Staubli VAL3: MFX_ROB_17.pjx

--- MFX_ROB_17.pjx ---
Parameters version=s7.9.1 stackSize=5000 millimeterUnit=true
Program file=checkAtPark.pgx
Program file=display.pgx
Program file=displayMessage.pgx
Program file=displayMessage1.pgx
Program file=displayMessage2.pgx
Program file=displayMessage3.pgx
Program file=displayMessage4.pgx
Program file=displayMessage5.pgx
Program file=displayMessage6.pgx
Program file=displayMessage7.pgx
Program file=displayMessage8.pgx
Program file=displayMessage9.pgx
Program file=initialize.pgx
Program file=initializeRobot.pgx
Program file=iocWriteBack.pgx
Program file=main.pgx
Program file=makePntAZELRA.pgx
Program file=mnuAdjTargetPnt.pgx
Program file=mnuEnterIPVals.pgx
Program file=mnuEnterTCPVals.pgx
Program file=mnuGetTCP.pgx
Program file=mnuGlobalSpeed.pgx
Program file=mnuMotionMenu.pgx
Program file=mnuMoveTargPnt.pgx
Program file=mnuMoveToPark.pgx
Program file=mnuSetTargetPts.pgx
Program file=mnuTeachCube.pgx
Program file=mnuTeachCyl.pgx
Program file=mnuTeachFrame.pgx
Program file=mnuTeachIP.pgx
Program file=mnuTeachMenu.pgx
Program file=mnuTeachPark.pgx
Program file=mnuTeachParkTop.pgx
Program file=mnuTeachSphere.pgx
Program file=mnuTeachStayClr.pgx
Program file=mnuTeachTCP.pgx
Program file=mnuTeachTCP4pnt.pgx
Program file=mnuTeachTCPptr.pgx
Program file=mnuTestSimESTOP.pgx
Program file=mnuUtility.pgx
Program file=movTargetPoint.pgx
Program file=movToPark.pgx
Program file=movToParkTop.pgx
Program file=readme.pgx
Program file=remCalcHere.pgx
Program file=remCalcHereSph.pgx
Program file=remCmdHandler.pgx
Program file=remDisableArm.pgx
Program file=remEnableArm.pgx
Program file=remEnableRem.pgx
Program file=remErrArgs.pgx
Program file=remErrBufferAdd.pgx
Program file=remErrBufferGet.pgx
Program file=remErrBusy.pgx
Program file=remErrCmd.pgx
Program file=remErrConfig.pgx
Program file=remErrFar.pgx
Program file=remErrInvalid.pgx
Program file=remErrManual.pgx
Program file=remErrNum.pgx
Program file=remErrPower.pgx
Program file=remErrPPTimeout.pgx
Program file=remErrRemoteKey.pgx
Program file=remErrTimeout.pgx
Program file=remErrZone.pgx
Program file=remGetArmStat.pgx
Program file=remGetDMOV.pgx
Program file=remGetESTOP.pgx
Program file=remGetHeartbeat.pgx
Program file=remGetHere.pgx
Program file=remGetHereSph.pgx
Program file=remGetIP.pgx
Program file=remGetIPVals.pgx
Program file=remGetJoints.pgx
Program file=remGetMaxA.pgx
Program file=remGetMaxDist.pgx
Program file=remGetMaxRV.pgx
Program file=remGetMaxV.pgx
Program file=remGetMode.pgx
Program file=remGetOneHere.pgx
Program file=remGetPPS.pgx
Program file=remGetRem.pgx
Program file=remGetRobotMode.pgx
Program file=remGetStagePos.pgx
Program file=remGetTCPVals.pgx
Program file=remGetWorld.pgx
Program file=remGetnGlobal.pgx
Program file=remMovAZELRA.pgx
Program file=remMovAxis.pgx
Program file=remMovBase.pgx
Program file=remMovHandler.pgx
Program file=remMovJoint.pgx
Program file=remMovJointAxis.pgx
Program file=remMovPoint.pgx
Program file=remMovSph.pgx
Program file=remMovSphAxis.pgx
Program file=remMovXYZ.pgx
Program file=remSetHeartbeat.pgx
Program file=remSetIP.pgx
Program file=remSetIPVals.pgx
Program file=remSetMaxA.pgx
Program file=remSetMaxDist.pgx
Program file=remSetMaxRV.pgx
Program file=remSetMaxV.pgx
Program file=remSetMode.pgx
Program file=remSetPPS.pgx
Program file=remSetStagePos.pgx
Program file=remSetTCPVals.pgx
Program file=remSetnGlobal.pgx
Program file=remTest.pgx
Program file=remTransIP.pgx
Program file=start.pgx
Program file=stop.pgx
Program file=tskCollision.pgx
Program file=tskHaltMoveMon.pgx
Program file=tskInterlocks.pgx
Program file=tskMonitorZone.pgx
Program file=tskRemControl1.pgx
Program file=tskSimESTOP.pgx
Data file=MFX_ROB_17.dtx
Library alias=io path=Disk://io/io.pjx autoload=true password=
Library alias=TCP4 path=Disk://calcTool4pEn/calcTool4pEn.pjx autoload=true password=
Library alias=MON path=Disk://monitorAreaEn/monitorAreaEn.pjx autoload=true password=

--- MFX_ROB_17.dtx ---
public bool bCubeStep1
public bool bCylinderStep1
bool bESTOPactive
public bool bEnableMonitor
public bool bInsideCube
public bool bInsideCylinder
public bool bInsideSphere
bool bKillRemControl
bool bMoveLinear = true
public bool bRemControlON
bool bRemMotionBusy
public bool bSetCubeXYZ
public bool bSetCylinderRZ
public bool bSetSphereRad
bool bSimESTOPOn
bool bSimulateESTOP
public bool bSphereStep1
public bool bStopAllMonitor = true
public bool bStopMotion
public bool bWatchForHalt
public bool bWorldFrameView = true
dio dCollisionSens = {link=usrIn0}
frame fIP1 = {fatherId=fIPoriginal[0]}
public frame fIP2 = {fatherId=fIPoriginal[0]}
frame fIPoriginal = {x=-1.16, y=-7.997692, z=1599.75028, rx=-90.079848, ry=0.325339, rz=-0.147005, fatherId=world[0]}
public jointRx jPark = {j1=89.588014, j2=-47.40785, j3=113.936199, j4=-0.155325, j5=-66.458795, j6=0.148711}
jointRx jParkTop = {j1=88.830052, j2=-90.553253, j3=149.996753, j4=-0.166481, j5=-59.375003, j6=0.928419}
mdesc mDefault = {accel=20, vel=20, decel=20, blend=off}
public mdesc mGlobalSpeed = {accel=20, vel=20, decel=20, blend=off}
mdesc mMdesc
public mdesc mSafeSlow = {accel=15, vel=20, decel=15, blend=off}
num nAccFast = 60
num nAccMedium = 40
num nAccSlow = 20
num nAdjPntMoveTol = 25
num nAzHere = -0.0000183783
num nColision = 1
num nDistXCube
num nDistYCube
num nDistZCube
num nDistZCylinder
num nElHere = 44.997695
num nErrBufferSize = 10
num nErrNext
num nErrNow
num nHeartbeat = 4344
num nIP1Azimuth[20]
  [1] = 45
  [2] = -45
  [3] = 45
  [4] = -45
  [5] = 9.38
  [6] = 7.44
  [7] = 17.53
  [8] = 48.36
  [9] = 142.53
  [10] = 140.2
  [11] = 145.08
  [12] = 142.4
  [13] = 142.23
  [14] = 144.96
  [15] = 106.35
  [16] = 100.36
  [17] = 19.8
  [18] = 8.88
  [19] = 23.034688
num nIP1Elevation[20]
  [3] = -45
  [4] = -45
  [5] = 21.19
  [6] = 39.23
  [9] = 37.74
  [10] = 30.33
  [11] = 44.59
  [12] = 42.45
  [13] = 38.39
  [14] = 44.81
  [15] = 29.56
  [16] = 45.35
  [17] = 29.88
  [18] = 12.25
  [19] = 8.727177
num nIP1Number = 1
num nIP1Radius[20]
  [1] = 600
  [2] = 600
  [3] = 600
  [4] = 600
  [5] = 1000
  [6] = 1000
  [7] = 300
  [8] = 250
  [9] = 300
  [10] = 300
  [11] = 300
  [12] = 300
  [13] = 300
  [14] = 300
  [15] = 300
  [16] = 300
  [17] = 100
  [18] = 200
  [19] = 857.27654
num nIP2Azimuth[20]
  [0] = 15
  [2] = -128.927
num nIP2Elevation[20]
  [0] = 20
  [2] = 79.165
num nIP2Number = 2
num nIP2Radius[20]
  [0] = 300
  [1] = 600
  [2] = 123.321
  [5] = 1000
num nIPNumber = -1
num nIdxAdjTargetPt = 291
num nIdxArmCalCheck = 31
num nIdxArmPowerOn = 181
num nIdxESTOPCheck = 121
num nIdxEnterIP = 341
num nIdxEnterTCP = 321
public num nIdxFrm1of5 = 131
public num nIdxFrm2of5 = 141
public num nIdxFrm3of5 = 151
public num nIdxFrm4of5 = 161
public num nIdxFrm5of5 = 171
num nIdxGetTCP = 351
public num nIdxMainMenu = 1
public num nIdxMotionMenu = 271
num nIdxMoveTargPt = 281
num nIdxMoveToPark = 311
num nIdxParkCheck = 41
public num nIdxPtrVerify
num nIdxRemControl = 321
public num nIdxResolution
public num nIdxSetCubeXYZ = 211
public num nIdxSetCylRZ = 231
num nIdxSetSpeeds = 181
public num nIdxSetSphRad = 251
num nIdxSetTargetPt = 261
public num nIdxStyClr = 61
public num nIdxTCP1of4 = 81
public num nIdxTCP2of4 = 91
public num nIdxTCP3of4 = 101
public num nIdxTCP4Point
public num nIdxTCP4of4 = 111
public num nIdxTeachClear
public num nIdxTeachCube = 201
public num nIdxTeachCyl = 221
num nIdxTeachIP = 331
public num nIdxTeachMenu = 11
public num nIdxTeachPARK = 51
num nIdxTeachPARKT = 371
public num nIdxTeachSph = 241
public num nIdxTeachTCP = 21
num nIdxUtilMenu2 = 301
num nIdxUtilityMenu = 71
num nMaxAccel = 50
num nMaxDist = 1000
num nMaxLoginTries = 3
num nMaxRVelo = 20
num nMaxVelo = 100
num nMovArgs
num nNumberCube
num nNumberCylinder
num nNumberSphere
num nPPS
num nParkTolerance = 50
num nRHere = 565.684578
num nRXHere = 0.0101053
num nRYHere = 0.000281961
num nRZHere = 0.00483895
num nRadiusCylinder
num nRadiusSphere
num nRemoteTimeout = 30
num nResolution[4]
  [0] = 0.001
  [1] = 0.01
  [2] = 0.1
  [3] = 1
num nRobotMode = 1
num nSelection = 1
num nStagePos
num nStagePosOK
num nVelFast = 60
num nVelMedium = 40
num nVelSlow = 20
num nXHere = -0.00012746
num nYHere = 399.983479
num nZHere = 400.0163407
num nZoneWatchTol = 25
public pointRx pCellReference = {shoulder=righty, elbow=epositive, wrist=wpositive, fatherId=world[0]}
pointRx pIP1NullPoint = {shoulder=sfree, elbow=efree, wrist=wfree, fatherId=fIP1[0]}
pointRx pIP1Point[20]
  [0] = {x=73, y=424, z=417, rx=-45, ry=-172, rz=-7, shoulder=sfree, elbow=efree, wrist=wfree, fatherId=fIP1[0]}
  [1] = {x=145, y=424, z=398, rx=-46, ry=-166, rz=-14, shoulder=sfree, elbow=efree, wrist=wfree, fatherId=fIP1[0]}
  [2] = {x=272, y=424, z=325, rx=-52, ry=-152, rz=-30, shoulder=sfree, elbow=efree, wrist=wfree, fatherId=fIP1[0]}
  [3] = {x=325, y=424, z=272, rx=-57, ry=-147, rz=-40, shoulder=sfree, elbow=efree, wrist=wfree, fatherId=fIP1[0]}
  [4] = {x=294, y=424, z=305, rx=-54, ry=-150, rz=-34, shoulder=sfree, elbow=efree, wrist=wfree, fatherId=fIP1[0]}
  [5] = {fatherId=fIP1[0]}
  [6] = {fatherId=fIP1[0]}
  [7] = {x=145, y=424, z=398, rx=-46, ry=-166, rz=-14, fatherId=fIP1[0]}
  [8] = {fatherId=fIP1[0]}
  [9] = {x=272, y=424, z=325, rx=-52, ry=-152, rz=-30, fatherId=fIP1[0]}
  [10] = {fatherId=fIP1[0]}
  [11] = {fatherId=fIP1[0]}
  [12] = {x=325, y=424, z=272, rx=-57, ry=-147, rz=-40, fatherId=fIP1[0]}
  [13] = {x=294, y=424, z=305, rx=-54, ry=-150, rz=-34, fatherId=fIP1[0]}
  [14] = {fatherId=fIP1[0]}
  [15] = {fatherId=fIP1[0]}
  [16] = {fatherId=fIP1[0]}
  [17] = {fatherId=fIP1[0]}
  [18] = {fatherId=fIP1[0]}
  [19] = {y=500, rx=90, rz=-180, fatherId=fIP1[0]}
pointRx pIP2NullPoint = {fatherId=fIP2[0]}
pointRx pIP2Point[20]
  [0] = {shoulder=sfree, elbow=efree, wrist=wfree, fatherId=fIP2[0]}
  [1] = {x=300, y=424.264069, z=300, rx=125.26439, ry=-30, rz=-35.26439, shoulder=sfree, elbow=efree, wrist=wfree, fatherId=fIP2[0]}
  [2] = {x=-300, y=424.264069, z=300, rx=125.26439, ry=30, rz=35.26439, shoulder=sfree, elbow=efree, wrist=wfree, fatherId=fIP2[0]}
  [3] = {x=300, y=-424.264069, z=300, rx=-125.26439, ry=-30, rz=35.26439, shoulder=sfree, elbow=efree, wrist=wfree, fatherId=fIP2[0]}
  [4] = {x=-300, y=-424.264069, z=300, rx=-125.26439, ry=30, rz=-35.26439, shoulder=sfree, elbow=efree, wrist=wfree, fatherId=fIP2[0]}
  [5] = {shoulder=sfree, elbow=efree, wrist=wfree, fatherId=fIP2[0]}
  [6] = {shoulder=sfree, elbow=efree, wrist=wfree, fatherId=fIP2[0]}
  [7] = {shoulder=sfree, elbow=efree, wrist=wfree, fatherId=fIP2[0]}
  [8] = {shoulder=sfree, elbow=efree, wrist=wfree, fatherId=fIP2[0]}
  [9] = {shoulder=sfree, elbow=efree, wrist=wfree, fatherId=fIP2[0]}
  [10] = {shoulder=sfree, elbow=efree, wrist=wfree, fatherId=fIP2[0]}
  [11] = {shoulder=sfree, elbow=efree, wrist=wfree, fatherId=fIP2[0]}
  [12] = {shoulder=sfree, elbow=efree, wrist=wfree, fatherId=fIP2[0]}
  [13] = {shoulder=sfree, elbow=efree, wrist=wfree, fatherId=fIP2[0]}
  [14] = {shoulder=sfree, elbow=efree, wrist=wfree, fatherId=fIP2[0]}
  [15] = {shoulder=sfree, elbow=efree, wrist=wfree, fatherId=fIP2[0]}
  [16] = {shoulder=sfree, elbow=efree, wrist=wfree, fatherId=fIP2[0]}
  [17] = {shoulder=sfree, elbow=efree, wrist=wfree, fatherId=fIP2[0]}
  [18] = {shoulder=sfree, elbow=efree, wrist=wfree, fatherId=fIP2[0]}
  [19] = {shoulder=sfree, elbow=efree, wrist=wfree, fatherId=fIP2[0]}
pointRx pMoveIP1Target = {fatherId=fIP1[0]}
pointRx pMoveIP2Target = {shoulder=sfree, elbow=efree, wrist=wfree, fatherId=fIP2[0]}
pointRx pMoveTarget = {shoulder=sfree, elbow=efree, wrist=wfree, fatherId=world[0]}
pointRx pNullPosition = {fatherId=world[0]}
pointRx pOriginCube = {fatherId=world[0]}
pointRx pOriginCylinder = {fatherId=world[0]}
pointRx pOriginSphere = {fatherId=world[0]}
pointRx teste[4]
  [0] = {x=7, y=243, z=26, rx=-4.03658e-18, ry=-79, rz=-9.47474e-33, shoulder=sfree, elbow=efree, wrist=wfree, fatherId=fIP1[0]}
  [1] = {x=17, y=243, z=28, rx=4.437099e-14, ry=-79.999286, rz=0.00497464, fatherId=fIP1[0]}
  [2] = {y=400, z=400, rx=0.01, ry=-2.827901e-23, rz=0.00516647, fatherId=fIP1[0]}
  [3] = {fatherId=fIP1[0]}
sio sioIOCclient = {link=Socket\MFX}
string sErrBuffer[10]
string sIOCCommand
string sIOCPassword = "USERPASSWORD"
string sIOCUserName = "CS8LOGIN"
string sIOCValue
string sIP1TargName[20]
  [0] = "v"
  [1] = "a"
  [2] = "sto 1"
  [3] = "ybco104"
  [4] = "cool oi"
  [5] = "magpeak2"
  [6] = "IP1 Point6 Name"
  [7] = "IP1 Point7 Name"
  [8] = "IP1 Point8 Name"
  [9] = "IP1 Point9 Name"
  [10] = "IP1 Point10 Name"
  [11] = "IP1 Point11 Name"
  [12] = "IP1 Point12 Name"
  [13] = "IP1 Point13 Name"
  [14] = "IP1 Point14 Name"
  [15] = "IP1 Point15 Name"
  [16] = "IP1 Point16 Name"
  [17] = "IP1 Point17 Name"
  [18] = "IP1 Point18 Name"
  [19] = "IP1 Point19 Name"
string sIP2TargName[20]
  [0] = "TestTeachPoint0"
  [1] = "IP2 Point1 Name"
  [2] = "IP2 Point2 Name"
  [3] = "IP2 Point3 Name"
  [4] = "IP2 Point4 Name"
  [5] = "a"
  [6] = "IP2 Point6 Name"
  [7] = "IP2 Point7 Name"
  [8] = "IP2 Point8 Name"
  [9] = "IP2 Point9 Name"
  [10] = "IP2 Point10 Name"
  [11] = "IP2 Point11 Name"
  [12] = "IP2 Point12 Name"
  [13] = "IP2 Point13 Name"
  [14] = "IP2 Point14 Name"
  [15] = "IP2 Point15 Name"
  [16] = "IP2 Point16 Name"
  [17] = "IP2 Point17 Name"
  [18] = "IP2 Point18 Name"
  [19] = "IP2 Point19 Name"
string sMenuBottomLine[53]
  [0] = " Tch. Mot. Util ---- ---- ---- ---- Stop"
  [1] = " Pnts IPCS Park ParkT TCP Zone  --- Ret."
  [2] = "RefP 4Pnt DEnt ---- ---- ---- ---- Ret."
  [3] = "---- ---- ---- Stop ---- ---- ---- Ret."
  [4] = "Cont ---- ---- Mov. ---- ---- ---- Ret."
  [5] = "Save ---- ---- ---- ---- ---- ---- Ret."
  [6] = "Cube Cyl. Sph. ---- ---- ---- ---- Ret."
  [7] = "Init Park Enbl Spds RemC TCP. ---- Ret."
  [8] = "Next ---- ---- ---- ---- ---- ---- Abrt"
  [9] = "Next ---- ---- ---- ---- ---- ---- Abrt"
  [10] = "Next ---- ---- ---- ---- ---- ---- Abrt"
  [11] = "Tch. ---- ---- ---- ---- ---- ---- Abrt"
  [12] = "Cont ---- ---- ---- ---- ---- ---- Abrt"
  [13] = "Next ---- Togl ---- ---- ---- ---- Abrt"
  [14] = "Next ---- ---- ---- ---- ---- ---- Abrt"
  [15] = "Next ---- ---- ---- ---- ---- ---- Abrt"
  [16] = "Next ---- ---- ---- ---- ---- ---- Abrt"
  [17] = "Save ---- ---- ---- ---- ---- ---- Abrt"
  [18] = "SVel MVel FVel ---- SAcc MAcc FAcc Ret."
  [20] = "Save ---- Chng Orig  XYZ ---- Clr. Ret."
  [21] = "Save ---- ----  DX   DY   DZ  ---- Ret."
  [22] = "Save ---- Chng Orig RadZ ---- Clr. Ret."
  [23] = "Save ---- ---- Rad.  DZ  ---- ---- Ret."
  [24] = "Save ---- Chng Orig Rad. ---- Clr. Ret."
  [25] = "Save ---- ---- Rad. ---- ---- ---- Ret."
  [26] = " IP  Pnt# Name Azi. Elev Rad.      Ret."
  [27] = "Pnts ---- ---- Park --- ParkTop -- Ret."
  [28] = " IP  Pnt# ---- ---- Adj. Mov. ---- Ret."
  [30] = "Init Park Dis. Spds RemC ---- ---- Ret."
  [31] = "Mov. ---- ---- ---- ---- ---- ---- Ret."
  [32] = " X    Y    Z    RX   RY   RZ  ---- Ret."
  [33] = "Sel. DEnt Wiz. ---- ---- ---- ---- Ret."
  [34] = " X    Y    Z    RX   RY   RZ  ---- Ret."
  [35] = " IP  ---- ---- ---- ---- ---- ---- Ret."
  [36] = "Cont ---- ---- ---- ---- ---- ---- Dis."
  [37] = "Save ---- ---- ---- ---- ---- ---- Ret."
string sNumConv = ".3"
string sRemMotionCmd
string sTargetChoice[3]
  [0] = "InteractionPoint1"
  [1] = "InteractionPoint2"
  [2] = "not "
public string sUserPageText[382]
  [0] = "(F1) (F2) (F3) (F4) (F5) (F6) (F7) (F8)"
  [1] = ">>  MAIN MENU  <<"
  [2] = "Select Your Choice...     (ESC aborts)"
  [3] = "TEACH MENU"
  [4] = "MOTION MENU"
  [5] = "UTILITY MENU"
  [10] = "END PROGRAM"
  [11] = ">>  TEACH MENU  <<"
  [12] = "Select Your Choice...     (ESC aborts)"
  [13] = "Teach TARGET POINTS"
  [14] = "Teach INTERACTION PNT COORD SYS"
  [15] = "Teach PARK Position"
  [16] = "Teach PARK TOP Position"
  [17] = "Teach TCP"
  [18] = "Teach STAY CLEAR ZONES"
  [20] = "RETURN"
  [21] = ">>  TEACH TCP  <<"
  [22] = "Select Your Choice...     (ESC aborts)"
  [23] = "Teach TCP w/ REF POINTER"
  [24] = "Teach TCP w/ 4-POINT METHOD"
  [25] = "TCP Values Direct Entry"
  [30] = "ABORT & RETURN"
  [31] = ">>  ARM NOT CALIBRATED!  <<"
  [32] = "MOTION NOT ALLOWED"
  [36] = "STOP PROGRAM"
  [40] = "ABORT & RETURN"
  [41] = ">>  VERIFY ARM AT PARK <<"
  [42] = "Select Your Choice...     (ESC aborts)"
  [46] = "Move to PARK"
  [50] = "ABORT & RETURN"
  [51] = ">>  TEACH PARK Position  <<"
  [52] = "               (ESC aborts)"
  [53] = "Instructions:"
  [54] = "1.  Change to MANUAL mode"
  [55] = "2.  Move robot to  PARK location"
  [59] = "(F1)  ACCEPT, SAVE, & RETURN"
  [60] = "(F8)  ABORT & RETURN"
  [61] = ">>  DEFINE STAY CLEAR ZONES  <<"
  [62] = "Select Your Choice...     (ESC aborts)"
  [63] = "CUBE Zones"
  [64] = "CYLINDER Zones"
  [65] = "SPHERE Zones"
  [70] = "ABORT & RETURN"
  [71] = ">>  UTILITY MENU  <<"
  [72] = "Select Your Choice...     (ESC aborts)"
  [73] = "Initialize Robot"
  [74] = "Verify Arm is at PARK location"
  [75] = "ENABLE  Zone Monitoring"
  [76] = "Set Global Speed Parameters"
  [77] = "Start IOC Client Remote Control"
  [78] = "Show Current TCP:IP Frame Vals"
  [80] = "RETURN"
  [81] = ">> TEACH TCP w/ Pointer:  1 of 4  <<"
  [82] = "               (ESC aborts)"
  [83] = "CONDITIONS REQD TO TEACH TCP"
  [84] = "#1:  Ref Pointer attached to Flange"
  [85] = "    (Defined tool = tRefPointer)"
  [86] = "#2:  Cell Ref Pointer in Workspace"
  [89] = "(F1)  CONTINUE to Step 2 of 4"
  [90] = "(F8)  ABORT & RETURN"
  [91] = ">>  TEACH TCP w/ Pointer:  2 of 4  <<"
  [92] = "               (ESC aborts)"
  [94] = "          MOVE ROBOT TO"
  [95] = "     CELL REFERENCE POINTER"
  [99] = "(F1)  CONTINUE to Step 3 of 4"
  [100] = "(F8)  ABORT & RETURN"
  [101] = ">>  TEACH TCP w/ Pointer:  3 of 4  <<"
  [102] = "               (ESC aborts)"
  [103] = "       DO THE FOLLOWING"
  [104] = "1.  REMOVE Reference Pointer Tool"
  [105] = "2.  ATTACH Sensor Tool"
  [106] = "3.  MOVE Sensor Tool to Cell Ref Ptr"
  [109] = "(F1) TEACH TOOL & CONTINUE"
  [110] = "(F8) ABORT & RETURN"
  [111] = ">>  TEACH TCP w/ Pointer:  4 of 4  <<"
  [112] = "               (ESC aborts)"
  [113] = "VERIFY the Sensor Tool Definition:"
  [114] = "1.  Switch to TOOL MODE on Pendant"
  [115] = "2.  Move  X, Y, Z, RX, RY, RZ "
  [116] = "  and verify motion"
  [119] = "(F1)  ACCEPT, SAVE,  AND RETURN"
  [120] = "(F8)  ABORT & RETURN WITHOUT SAVE"
  [121] = ">>  ESTOP CHECK <<"
  [122] = "Select Your Choice...     (ESC aborts)"
  [123] = "(F1)  Continue"
  [130] = "(F8)  ABORT & RETURN"
  [131] = ">>  TEACH IP COORD SYS:  1 of 5  <<"
  [132] = "               (ESC aborts)"
  [134] = "SELECT IP COORD SYS TO TEACH"
  [136] = "(F1)  ACCEPT & CONTINUE"
  [138] = "(F3)  Toggle INT POINT CS Selection"
  [140] = "(F8)  ABORT & RETURN"
  [141] = ">>  TEACH INT POINT CS:  2 of 5  <<"
  [142] = "               (ESC aborts)"
  [145] = "ATTACH REF POINTER"
  [146] = "TO ROBOT FLANGE"
  [149] = "(F1)  CONTINUE"
  [150] = "(F8)  ABORT & RETURN"
  [151] = ">>  TEACH INT POINT CS:  3 of 5  <<"
  [152] = "               (ESC aborts)"
  [155] = "MOVE  REF POINTER TO"
  [156] = "INTERATION POINT COORD SYS"
  [157] = "ORIGIN POINT"
  [159] = "(F1)  CONTINUE"
  [160] = "(F8)  ABORT & RETURN"
  [161] = ">>  TEACH INT POINT CS:  4 of 5  <<"
  [162] = "               (ESC aborts)"
  [165] = "MOVE REF POINTER TO"
  [166] = "INTERACTION POINT COORD SYS"
  [167] = "X-AXIS POINT"
  [169] = "(F1)  CONTINUE"
  [170] = "(F8)  ABORT & RETURN"
  [171] = ">>  TEACH INT POINT CS:  5 of 5  <<"
  [172] = "               (ESC aborts)"
  [175] = "MOVE REF POINTER TO"
  [176] = "INTERACTION POINT COORD SYS"
  [177] = "Y-AXIS POINT"
  [179] = "(F1)  ACCEPT, SAVE,  & RETURN"
  [180] = "(F8)  ABORT & RETURN WITHOUT SAVE"
  [181] = ">>  SET GLOBAL SPEED PARMS  <<"
  [182] = "Select Your Choice...     (ESC aborts)"
  [183] = "Slow Speed"
  [184] = "Medium Speed"
  [185] = "Fast Speed"
  [187] = "Slow Accel"
  [188] = "Medium Accel"
  [189] = "Fast Accel"
  [190] = "Return"
  [191] = ">>  TEACH PARK Position  <<"
  [192] = "               (ESC aborts)"
  [193] = "Move to PARK Position, F1 to continue..."
  [200] = "GO BACK"
  [201] = ">>  DEFINE CUBE Stay Clear Zone  <<"
  [202] = "               (ESC aborts)"
  [204] = "(F1)  ACCEPT, SAVE, & RETURN"
  [206] = "(F3)  Change Cube Number"
  [207] = "(F4)  Teach Cube Origin Point"
  [208] = "(F5)  Define DX, DY, DZ"
  [209] = "(F7)  Clear This Cube Definition"
  [210] = "(F8)  ABORT & RETURN"
  [211] = ">>  SET CUBE DX DY DZ <<"
  [212] = "               (ESC aborts)"
  [215] = "(F1)  ACCEPT DX/DY/DZ VALUES"
  [216] = "(F4)  Enter New DX Value"
  [217] = "(F5)  Enter New DY Value"
  [218] = "(F6)  Enter New DZ Value"
  [220] = "(F8)  ABORT & RETURN"
  [221] = ">>  DEFINE CYLINDER Stay Clear Zone  <<"
  [222] = "               (ESC aborts)"
  [224] = "(F1)  ACCEPT, SAVE, & RETURN"
  [226] = "(F3)  Change Cylinder Number"
  [227] = "(F4)  Teach Cylinder Origin Point"
  [228] = "(F5)  Define Cylinder Radius & DZ"
  [229] = "(F7)  Clear this Cylinder Definition"
  [230] = "(F8)  ABORT & RETURN"
  [231] = ">>  SET CYLINDER RAD & DZ  <<"
  [232] = "               (ESC aborts)"
  [235] = "(F1)  ACCEPT RAD/DZ VALUES"
  [236] = "(F4)  Enter New RADIUS Value"
  [237] = "(F5)  Enter New DZ Value"
  [240] = "(F8)  ABORT & RETURN"
  [241] = ">>  DEFINE SPHERE Stay Clear Zone  <<"
  [242] = "               (ESC aborts)"
  [244] = "(F1)  ACCEPT, SAVE, & RETURN"
  [246] = "(F3)  Change Sphere Number"
  [247] = "(F4)  Teach Sphere Origin Point"
  [248] = "(F5)  Define Sphere Radius"
  [249] = "(F7)  Clear This Sphere Definition"
  [250] = "(F8)  ABORT & RETURN"
  [251] = ">>  SET SPHERE RADIUS  <<"
  [252] = "               (ESC aborts)"
  [255] = "(F1)  ACCEPT RADIUS VALUE"
  [256] = "(F4)  Enter New RADIUS Value"
  [260] = "(F8)  ABORT & RETURN"
  [261] = ">>  SET TARGET POINTS  <<"
  [262] = "(F1) IP Nbr      :"
  [263] = "(F2) Pnt Nbr     :"
  [264] = "(F3) Name        :"
  [265] = "(F4) Azimuth     :"
  [266] = "(F5) Elevation   :"
  [267] = "(F6) Radius      :"
  [268] = "     X:         Y:         Z:"
  [269] = "    RX:        RY:        RZ:"
  [270] = "(F8)  SAVE, UPDATE, & RETURN"
  [271] = ">>  MOTION MENU  <<"
  [272] = "Select Your Choice...     (ESC aborts)"
  [273] = "Move & Adjust TARGET POINTS"
  [276] = "Move to PARK POSITION"
  [278] = "Move to PARK TOP POSITION"
  [280] = "ABORT"
  [281] = ">>  MOVE & ADJUST TARGET POINTS  <<"
  [282] = "(F1) IP Nbr      :"
  [283] = "(F2) Pnt Nbr     :"
  [284] = "        Name        :"
  [285] = "       Azimuth     :"
  [286] = "       Elevation   :"
  [287] = "       Radius      :"
  [288] = "     X:         Y:         Z:"
  [289] = "    RX:        RY:        RZ:"
  [290] = "(F6) MOVE TO   (F8) ABORT & RETURN"
  [291] = ">>  ADJUST TARGET POINTS  <<"
  [296] = "  Resolution:"
  [297] = "  Target RX:"
  [298] = "  Target RY:"
  [299] = "  Target RZ:"
  [301] = ">>  UTILITY MENU  <<"
  [302] = "Select Your Choice...     (ESC aborts)"
  [303] = "Initialize Robot"
  [304] = "Verify Arm is at PARK location"
  [305] = "DISABLE Zone Monitoring"
  [306] = "Set Global Speed Parameters"
  [307] = "Start IOC Host Remote Control"
  [310] = "RETURN"
  [311] = ">>  MOVE TO  PARK  <<"
  [312] = "Select Your Choice...     (ESC aborts)"
  [313] = "Start Move to PARK Location"
  [320] = "ABORT"
  [321] = ">>  DIRECT ENTRY TCP VALUES  <<"
  [322] = " Enter Values...        ESC Aborts"
  [323] = " TCP-X"
  [324] = " TCP-Y"
  [325] = " TCP-Z"
  [326] = " TCP-RX"
  [327] = " TCP-RY"
  [328] = " TCP-RZ"
  [330] = " F8 = Save & Return"
  [331] = ">> TEACH INTERATION PNTS <<"
  [332] = "Select Your Choice...       ESC Aborts"
  [333] = "(F1)  Select Interaction Point"
  [334] = "(F2)  Direct Entry of IP Data"
  [335] = "(F3)  Run IP Teach Wizard"
  [337] = "(F8)  Return"
  [341] = ">>  DIRECT ENTRY IP VALUES  <<"
  [342] = " Enter Values...        ESC Aborts"
  [343] = "IP-X"
  [344] = "IP-Y"
  [345] = "IP-Z"
  [346] = "IP-RX"
  [347] = "IP-RY"
  [348] = "IP-RZ"
  [350] = "(F8)  Save & Return"
  [351] = ">>  DISPLAY TCP VALUES @ IP  <<"
  [352] = "                        ESC Aborts"
  [353] = "Current IP  :"
  [354] = "TCP.x       :"
  [355] = "TCP.y       :"
  [356] = "TCP.z       :"
  [357] = "TCP.rx      :"
  [358] = "TCP.ry      :"
  [359] = "TCP.rz      :"
  [361] = ">>  STARTUP CHECK 0UT  <<"
  [363] = "WARNING:  ESTOP Simulation = ACTIVE !"
  [365] = "F1:  CONTINUE"
  [367] = "F8:  Disable ESTOP Simulation"
  [370] = "ABORT & RETURN"
  [371] = ">>  TEACH PARK Position  <<"
  [372] = "               (ESC aborts)"
  [373] = "Instructions:"
  [374] = "1.  Change to MANUAL mode"
  [375] = "2.  Move robot to  PARK TOP location"
tool tNULLTOOL = {fatherId=flange[0], ioLink=valve1}
public tool tRefPointer = {fatherId=flange[0], ioLink=valve1}
tool tSensorTool = {z=162.433, ry=90, rz=-90, fatherId=flange[0], ioLink=valve1}
trsf trUserTool

--- main.pgx ---
public program main()
  local bool LbStopProgram
  local joint LjHere
  local num LnAcknowledge
  local num LnDistance
  local point LpHere
  local point LpPark
  local point LpTargetPoint
  local num nKey
begin
  //header begin
  // PROGRAM main()
  //
  // runs the entire application
  // menus
  // mode control
  //
  // incoming parms:  none
  // outgoing parms:  none
  // called from:  pgm start()
  //
  //  NOTE:  the strings structure is in groups of 10 in the strings array sUserPageText[ ]
  //
  //  initial release KN
  //header end
  //
  // initialize important variables & parameters
  call initialize()
  //
  // test for bSimulateESTOP is true, announce to user if so
  call mnuTestSimESTOP()
  //
  // start the ESTOP Monitoring task
  //taskCreate "MonitorESTOP",25,tskMonitorESTOP()
  // initialize robot (ESTOP=off, POWER=on, Arm=CALIBRATED)
  call initializeRobot()
  //
  // start the task to enable/disable Stay Clear Zone monitoring
  taskCreate "MonitorZone",10,tskMonitorZone()
  //
  // start the IOC Host communications task
  // enabled from Utility Menu calls & operator input
  // HALTed by command from IOC host
  // killed on stop()
  //taskCreate "RemoteControl",40,tskRemControl()
  // MC used a different version of tskRemControl that does not look for remote mode
  sioCtrl(io:IOC,"timeout",0)
  taskCreate "RemoteControl",40,tskRemControl1()

  taskCreate "Interlocks",40,tskInterlocks()
  taskCreate "Colision Sensor",40,tskCollision()

  //
  // start the task that will be used to monitor a MCP keypress command to halt robot motion during manual mode
  taskCreate "MonitorHalt",20,tskHaltMoveMon()
  //
  // check if arm is at pre-defined jPark location, advise user if not but do not force action
  // get current position, compare with destination
  LpHere=here(tSensorTool,world)
  LpPark=jointToPoint(tSensorTool,world,jPark)
  LnDistance=abs(distance(LpHere,LpPark))
  if LnDistance>nParkTolerance
    popUpMsg("WARNING  WARNING  WARNING  WARNING       Arm is NOT PARKED")
  endIf

  if nStagePos!=nStagePosOK
    popUpMsg("Z stage not at interation zone. Robot will not power.")
  endIf
  //
  // start infinite loop to run application
  // halts on operator command
  LbStopProgram=false
  do
    // nIdxMainMenu=1
    call display(nIdxMainMenu,nKey)

    if nStagePos!=nStagePosOK
      popUpMsg("Z stage not at interation zone. Robot will not power.")
    endIf

    // verify selection
    switch nKey
      // ESC not allowed at MAIN MENU...must use F8=STOP Program
      case 255
        //
      break
      // menu = Main Menu:  F1 Button, change to TEACH menu
      case 271
        call mnuTeachMenu()
      break
      // menu = Main Menu:  F2 Button, change to MOTION menu
      case 272
        call mnuMotionMenu()
      break
      // menu = Main Menu:  F3 Button, change to UTILITY menu
      case 273
        call mnuUtility()
      break
      // menu = Main Menu:  F8 Button, End Application & Exit
      case 278
        LbStopProgram=true
      break
      // ALL OTHER CHOICES
      default
        popUpMsg("BAD SELECTION...Press OK")
      break
    endSwitch
  until (false or (LbStopProgram==true))
  call stop()
  // done
end

--- start.pgx ---
program start()
  local joint jNew
  local mdesc l_mMdesc
  local point l_pAxisOx
  local point l_pOrigin
  local point l_pPlaneOxy
  local num nKey
begin
  //-----------------------------------------------------------------------
  //Header begin
  //Description of program
  //
  //
  //History
  //  Initial Release KN
  //Header end
  //-----------------------------------------------------------------------
  // Global variables :
  //
  //---------------------
  //start description
  //---------------------


  //  l_pOrigin = {{-1.15694092, -7.99769233,  1599.75028 , 0 ,0 ,0}, {sfree,efree,wfree}}
  //  l_pAxisOx = {{38.8422826, -8.22467660,  1599.85322 , 0 ,0 ,0}, {sfree,efree,wfree}}
  //  l_pPlaneOxy = {{38.9449094, -8.28100326,  1559.85339 , 0 ,0 ,0}, {sfree,efree,wfree}}
  //  link(l_pOrigin,world)
  //  link(l_pAxisOx,world)
  //  link(l_pPlaneOxy,world)

  //  setFrame(l_pOrigin,l_pAxisOx,l_pPlaneOxy,fCalculatedFram)

  //  logMsg("x  "+toString(".6",fCalculatedFram.trsf.x))
  //  logMsg("y  "+toString(".6",fCalculatedFram.trsf.y))
  //  logMsg("z  "+toString(".6",fCalculatedFram.trsf.z))
  //  logMsg("rx "+toString(".6",fCalculatedFram.trsf.rx))
  //  logMsg("ry "+toString(".6",fCalculatedFram.trsf.ry))
  //  logMsg("rz" +toString(".6",fCalculatedFram.trsf.rz))

  if (false)

    if (pointToJoint(tSensorTool,jPark,teste[1],jNew))
      logMsg("bom")
    else
      logMsg("mau")
    endIf

    // movel(pIP1Point[nIP1Number],tSensorTool,mGlobalSpeed)
    //movel(pIP1Point[nIP1Number],tSensorTool,mGlobalSpeed)



    enablePower()

    do
      nKey=getKey()
      switch nKey
        // ESC key aborts & returns immediately
        case 271
          stopMove()
          resetMotion()
          movej(jPark,tSensorTool,mDefault)


        break
        case 272



          stopMove()
          resetMotion()
          movel(pIP1Point[0],tSensorTool,mDefault)

        break
        case 273


          stopMove()
          resetMotion()
          movel(pIP1Point[1],tSensorTool,mDefault)

          logMsg("x  "+toString(".6",teste[1].trsf.x))
          logMsg("y  "+toString(".6",teste[1].trsf.y))
          logMsg("z  "+toString(".6",teste[1].trsf.z))
          logMsg("rx "+toString(".6",teste[1].trsf.rx))
          logMsg("ry "+toString(".6",teste[1].trsf.ry))
          logMsg("rz"+toString(".6",teste[1].trsf.rz))
        break
        case 274
          stopMove()
          resetMotion()
          movel(pIP1Point[2],tSensorTool,mDefault)
        break
        case 275
          stopMove()
          resetMotion()
          movel(pIP1Point[3],tSensorTool,mDefault)
        break
        case 276
          stopMove()
          resetMotion()
          movel(pIP1Point[4],tSensorTool,mDefault)
        break
        case 277
          stopMove()
          resetMotion()
          movel(pIP1Point[5],tSensorTool,mDefault)
        break

        default
          //popUpMsg("errado")
        break

      endSwitch

    until (nKey==278)

    stopMove()
    resetMotion()
    //  enablePower()



    popUpMsg("fim")

  endIf



  call main()
end

--- checkAtPark.pgx ---
program checkAtPark()
  local bool LbParkContinue
  local point LpHere
  local num nKey
begin
  //header begin
  // PROGRAM checkAtPark()
  //
  // checks for Arm is at Park position
  //
  // incoming parms:  none
  // outgoing parms:  none
  // called from:  pgm mnuUtility()
  //
  //  initial release KN
  //header end
  //
  // clear motion stack of all movement commands
  stopMove()
  resetMotion()
  //
  userPage()
  cls()
  //
  // Verify arm is at PARK location.  Use pgm display() for menu control.
  // No motion except RX, RY, RZ adjustments can be made unless starting motion at PARK.
  // If arm is >nParkTolerance from PARK, user must move arm or abort.
  LpHere=here(tSensorTool,world)
  //
  //
  LbParkContinue=false
  do
    // nIdxParkCheck=41
    call displayMessage4(nIdxParkCheck,nKey)
    // verify selection
    switch nKey
      // ESC key aborts & returns immediately to previous menu
      case 255
        return
      break
      // Arm Park Check:  F4 to move to PARK position
      case 274
        call movToPark()
      break
      // Arm Park Check:  Abort & return immediately to previous menu
      case 278
        return
      break
      // Any other key press
      default
        popUpMsg("BAD SELECTION...press OK")
      break
    endSwitch
  until (false or (LbParkContinue==true))
  // done
end

--- display.pgx ---
program display(num nTitle (dimensions=1), num& nKey[] (dimensions=1))
  local bool LbKey
  local num LnFirst
  local num LnIndex
  local num LnQuestion
begin
  //header begin
  // PROGRAM display(nTitle, nKey)
  //
  // generic pgm used for menu displays and selection handling
  //
  // input parms:
  //    nTitle = index of selected menu Title string in sUserPageText[ ]
  //
  // other parms:
  //    nQuestion = index of selected menu Question string in sUserPageText[ ]
  //    nFirst = index of the first menu Items to be displayed from sUserPageText[ ]
  //
  //  NOTE:  the strings structure is in groups of 10 in the strings array sUserPageText[ ]
  //  Menu Page Indices are NUMBER variables
  //
  // output parms:
  //    nKey = the keypad number of the selected Function Key
  //
  // called from:  various
  // initial release KN
  //header end
  //
  // init local variables used as menu string text pointers
  // values are simply +1 & +2 offset of nTitle pointer
  LnQuestion=nTitle+1
  LnFirst=nTitle+2
  // clear user page and throw a title
  userPage()
  cls()
  title(sUserPageText[nTitle])
  //
  // print the F1 thru F8 Function Button Identifiers
  // at bottom of user window
  gotoxy(0,13)
  // bottom line text is indexed with respect to sUserPageText[]
  put(sMenuBottomLine[(nTitle-1)/10])
  //
  //print QUESTION or COMMAND
  gotoxy(0,1)
  put(sUserPageText[LnQuestion])
  //
  // print eight (F-) function identifiers & text on left hand side of userPage window
  for LnIndex=LnFirst to LnFirst+7
    gotoxy(1,LnIndex-LnFirst+3)
    put("(F")
    put(toString("",LnIndex-LnFirst+1))
    put(") ")
    put(sUserPageText[LnIndex])
  endFor
  //
  // Wait indefinitely for a function button press
  LbKey=false
  getKey()
  do
    nKey=getKey()
    switch nKey
      // ESC character always ABORTS AND/OR RETURNS
      case 255
        LbKey=true
      break
      case 271,272,273,274,275,276,277,278
        LbKey=true
      break
    endSwitch
    //
    delay(0)
  until (LbKey==true)
end

--- displayMessage.pgx ---
program displayMessage(num nTitle (dimensions=1), num& nKey[] (dimensions=1))
  local bool LbKey
  local num LnFirst
  local num LnIndex
  local num LnQuestion
begin
  //header begin
  // program displayMessage(nTitle, nKey)
  //
  // generic pgm used for displaying complex messages and reacting to user keypad selections
  // (this program modified from pgm display( )
  //
  // input parms:
  //    nTitle = index of selected menu Title string in sUserPageText[ ]
  //
  // other parms:
  //    nQuestion = nTitle+1 = index of selected menu Question string in sUserPageText[ ]
  //    nFirst = nTitle+2 = index of the first menu Items to be displayed from sUserPageText[ ]
  //
  //  NOTE:  the strings structure is in groups of 10 in the strings array sUserPageText[ ]
  //  Menu Page Indices are NUMBER variables
  //
  // output parms:
  //    nKey = the keypad number of the selected Function Key
  //
  // called from:  various
  // initial release KN
  //header end
  //
  // init local variables used as menu string text pointers
  // values are just +1 & +2 offset of nTitle pointer
  LnQuestion=nTitle+1
  LnFirst=nTitle+2
  // clear user page, and throw a title
  userPage()
  cls()
  title(sUserPageText[nTitle])
  //
  // Print menu page Function Button Identifiers at bottom of user window
  gotoxy(0,13)
  put(sMenuBottomLine[(nTitle-1)/10])
  //
  //print QUESTION or COMMAND
  gotoxy(0,2)
  put(sUserPageText[LnQuestion])
  //
  // print 8 statements from menu string data
  for LnIndex=LnFirst to LnFirst+7
    gotoxy(0,LnIndex-LnFirst+3)
    put(sUserPageText[LnIndex])
  endFor
  //
  // print the TargetChoice variable for Frame Teach
  gotoxy(0,0)

  if nIPNumber==-1
    put("ACTIVE IP = Original hutch IP")
  else
    put("ACTIVE IP = "+sTargetChoice[nIPNumber])
  endIf
  // Wait indefinitely for a function button press
  LbKey=false
  getKey()
  do
    nKey=getKey()
    switch nKey
      // ESC key always ABORTS AND / OR RETURNS
      case 255
        LbKey=true
      break
      // Function Button value returned for selected action
      case 271,272,273,274,275,276,277,278
        LbKey=true
      break
    endSwitch
    //
    delay(0)
  until (LbKey==true)
end

--- displayMessage1.pgx ---
program displayMessage1(num nTitle (dimensions=1), num& nKey[] (dimensions=1))
  local bool LbKey
  local num LnFirst
  local num LnIndex
  local num LnQuestion
begin
  //header begin
  // program displayMessage1(nTitle, nKey)
  //
  // generic pgm used for displaying complex messages and reacting to user keypad selections
  // (this program modified from pgm display( )
  //  CUSTOMIZED SPECIFICALLY FOR CUBE/CYL/SPHERE STAY CLEAR AREA DEFINITION
  //
  // input parms:
  //    nTitle = index of selected menu Title string in sUserPageText[ ]
  //
  // other parms:
  //    nQuestion = nTitle+1 = index of selected menu Question string in sUserPageText[ ]
  //    nFirst = nTitle+2 = index of the first menu Items to be displayed from sUserPageText[ ]
  //
  //  NOTE:  the strings structure is in groups of 10 in the strings array sUserPageText[ ]
  //  Menu Page Indices are NUMBER variables
  //
  // output parms:
  //    nKey = the keypad number of the selected Function Key
  //
  // called from:  various
  //
  // initial release KN
  //header end
  //
  // init local variables used as menu string text pointers
  // values are just +1 & +2 offset of nTitle pointer
  LnQuestion=nTitle+1
  LnFirst=nTitle+2
  // clear user page, and throw a title
  userPage()
  cls()
  title(sUserPageText[nTitle])
  //
  // print the user page Function Button Identifiers at bottom of page
  gotoxy(0,13)
  put(sMenuBottomLine[(nTitle-1)/10])
  //
  //print QUESTION or COMMAND
  gotoxy(0,1)
  put(sUserPageText[LnQuestion])
  //
  // print 8 statements from menu string data
  for LnIndex=LnFirst to LnFirst+7
    gotoxy(0,LnIndex-LnFirst+3)
    put(sUserPageText[LnIndex])
  endFor
  //
  // special setup for cube teach step 1
  if (bCubeStep1==true)
    // print current cube number
    gotoxy(0,0)
    put("Cube Number= ")
    put(toString(".0",nNumberCube))
    // print cube zone status
    gotoxy(19,0)
    put("Status=")
    if MON:bCreateCube[nNumberCube]==true
      put("DEFINED")
    else
      put("UNDEFINED")
    endIf
    // print cube Origin X, Y, Z
    gotoxy(0,1)
    put("Origin( ")
    put(toString("5.0",pOriginCube.trsf.x))
    put(", ")
    put(toString("5.0",pOriginCube.trsf.y))
    put(", ")
    put(toString("5.0",pOriginCube.trsf.z))
    put(" )")
    // print DX, DY, DZ
    gotoxy(0,2)
    put("DX= ")
    put(toString("5.0",nDistXCube))
    put(" DY= ")
    put(toString("5.0",nDistYCube))
    put(" DZ= ")
    put(toString("5.0",nDistZCube))
  endIf
  //
  // Special setup for Cube DX, DY, DZ
  if (bSetCubeXYZ==true)
    // print current cube number
    gotoxy(0,0)
    put("Cube Number= ")
    put(toString(".0",nNumberCube))
    // print cube zone status
    gotoxy(19,0)
    put("Status=")
    if MON:bCreateCube[nNumberCube]==true
      put("DEFINED")
    else
      put("UNDEFINED")
    endIf
    // print DX, DY, DZ
    gotoxy(0,1)
    put("DX=")
    put(toString("5.0",nDistXCube))
    gotoxy(0,2)
    put("DY=")
    put(toString("5.0",nDistYCube))
    gotoxy(0,3)
    put("DZ=")
    put(toString("5.0",nDistZCube))
  endIf
  //
  // special setup for cylinder teach step 1
  if (bCylinderStep1==true)
    // print current cylinder number
    gotoxy(0,0)
    put("Cyl Number= ")
    put(toString(".0",nNumberCylinder))
    // print cylinder zone status
    gotoxy(19,0)
    put("Status=")
    if MON:bCreateCylinder[nNumberCylinder]==true
      put("DEFINED")
    else
      put("UNDEFINED")
    endIf
    // print cylinder Origin X, Y, Z
    gotoxy(0,1)
    put("Origin( ")
    put(toString("5.0",pOriginCylinder.trsf.x))
    put(", ")
    put(toString("5.0",pOriginCylinder.trsf.y))
    put(", ")
    put(toString("5.0",pOriginCylinder.trsf.z))
    put(" )")
    // print cylinder Radius & DZ
    gotoxy(0,2)
    put("RAD = ")
    put(toString("5.0",nRadiusCylinder))
    put(" DZ = ")
    put(toString("5.0",nDistZCylinder))
  endIf
  //
  // Special setup for Cylinder Radius & DZ
  if (bSetCylinderRZ==true)
    // print current cylinder number
    gotoxy(0,0)
    put("Cyl Number= ")
    put(toString(".0",nNumberCylinder))
    // print cylinder zone status
    gotoxy(19,0)
    put("Status=")
    if MON:bCreateCylinder[nNumberCylinder]==true
      put("DEFINED")
    else
      put("UNDEFINED")
    endIf
    // print cylinder Radius & DZ
    gotoxy(0,1)
    put("RAD =")
    put(toString("5.0",nRadiusCylinder))
    gotoxy(0,2)
    put("DZ =")
    put(toString("5.0",nDistZCylinder))
  endIf
  //
  // special setup for sphere teach step 1
  if (bSphereStep1==true)
    // print current sphere number
    gotoxy(0,0)
    put("Sphere Number = ")
    put(toString(".0",nNumberSphere))
    // print sphere zone status
    gotoxy(19,0)
    put("Status=")
    if MON:bCreateSphere[nNumberSphere]==true
      put("DEFINED")
    else
      put("UNDEFINED")
    endIf
    // print sphere Origin X, Y, Z
    gotoxy(0,1)
    put("Origin( ")
    put(toString("5.0",pOriginSphere.trsf.x))
    put(", ")
    put(toString("5.0",pOriginSphere.trsf.y))
    put(", ")
    put(toString("5.0",pOriginSphere.trsf.z))
    put(" )")
    // print sphere Radius
    gotoxy(0,2)
    put("RAD = ")
    put(toString("5.0",nRadiusSphere))
  endIf
  //
  // Special setup for sphere Radius
  if (bSetSphereRad==true)
    // print current cylinder number
    gotoxy(0,0)
    put("Sphere Number= ")
    put(toString(".0",nNumberSphere))
    // print sphere zone status
    gotoxy(19,0)
    put("Status=")
    if MON:bCreateSphere[nNumberSphere]==true
      put("DEFINED")
    else
      put("UNDEFINED")
    endIf
    // print sphere Radius
    gotoxy(0,1)
    put("RAD =")
    put(toString("5.0",nRadiusSphere))
  endIf
  //
  // Wait indefinitely for a function button press
  LbKey=false
  getKey()
  do
    nKey=getKey()
    switch nKey
      // ESC character always ABORTS AND/OR RETURNS
      case 255
        LbKey=true
      break
      case 271,272,273,274,275,276,277,278
        LbKey=true
      break
    endSwitch
    //
    delay(0)
  until (LbKey==true)
end

--- displayMessage2.pgx ---
program displayMessage2(num nTitle (dimensions=1), num& nKey[] (dimensions=1))
  local bool LbKey
  local num LnFirst
  local num LnIndex
  local num LnQuestion
  local trsf LtrDisplay
begin
  //header begin
  // program displayMessage2(nTitle, nKey)
  //
  // generic pgm used for displaying complex messages and reacting to user keypad selections
  // (this program modified from pgm display( )
  //  CUSTOMIZED SPECIFICALLY FOR TARGET FRAME / TARGET POINT DEFINITION
  //  WITH AZIMUTH-ELEVATION-RADIUS CONVERSION TO X,Y,Z,RX,RY,RZ
  //
  // input parms:
  //    nTitle = index of selected menu Title string in sUserPageText[ ]
  //
  // other parms:
  //    nQuestion = nTitle+1 = index of selected menu Question string in sUserPageText[ ]
  //    nFirst = nTitle+2 = index of the first menu Items to be displayed from sUserPageText[ ]
  //
  //  NOTE:  the strings structure is in groups of 10 in the strings array sUserPageText[ ]
  //  Menu Page Indices are NUMBER variables
  //
  // output parms:
  //    nKey = the keypad number of the selected Function Key
  //
  // called from:  pgm  setTargetPts()
  // initial release KN
  //
  //header end
  //
  // init local variables used as menu string text pointers
  // values are simply +1 & +2 offset of nTitle pointer
  LnQuestion=nTitle+1
  LnFirst=nTitle+2
  // clear user page, and throw a title
  userPage()
  cls()
  title(sUserPageText[nTitle])
  //
  // print the Function Button Identifiers at bottom of page
  // selection uses pattern of one menu every 10 lines in sUserPageText[]
  gotoxy(0,13)
  put(sMenuBottomLine[(nTitle-1)/10])
  //
  // put the view change button on F7 to display coordinates relative to World or IP
  gotoxy(29,12)
  put("Frame")
  gotoxy(30,13)
  if bWorldFrameView==true
    put("Wrld")
  else
    put(" IP ")
  endIf
  //
  gotoxy(0,0)
  put("  F-Key to edit, ESC aborts edit")
  gotoxy(0,1)
  put(sUserPageText[nTitle+1])
  gotoxy(0,2)
  put(sUserPageText[nTitle+2])
  gotoxy(0,3)
  put(sUserPageText[nTitle+3])
  gotoxy(0,4)
  put(sUserPageText[nTitle+4])
  gotoxy(0,5)
  put(sUserPageText[nTitle+5])
  gotoxy(0,6)
  put(sUserPageText[nTitle+6])
  gotoxy(0,8)
  put(sUserPageText[nTitle+7])
  gotoxy(0,9)
  put(sUserPageText[nTitle+8])
  gotoxy(0,11)
  put(sUserPageText[nTitle+9])
  // print Target/Frame Number
  gotoxy(18,1)
  put(toString("",nIPNumber)+" = "+sTargetChoice[nIPNumber])
  // print number of selected Interaction Point
  gotoxy(18,2)
  if nIPNumber==0
    put(toString("",nIP1Number))
  else
    put(toString("",nIP2Number))
  endIf
  // print Name string of selected Interaction Point
  gotoxy(19,3)
  if nIPNumber==0
    put(sIP1TargName[nIP1Number])
  else
    put(sIP2TargName[nIP2Number])
  endIf
  // print Azimuth of selected Interaction Point & Target Point
  gotoxy(19,4)
  if nIPNumber==0
    put(toString(".3",nIP1Azimuth[nIP1Number]))
  else
    put(toString(".3",nIP2Azimuth[nIP2Number]))
  endIf
  // print Elevation of selected Interaction Point & Target Point
  gotoxy(19,5)
  if nIPNumber==0
    put(toString(".3",nIP1Elevation[nIP1Number]))
  else
    put(toString(".3",nIP2Elevation[nIP2Number]))
  endIf
  // print Radius of selected Interaction Point & Target Point
  gotoxy(19,6)
  if nIPNumber==0
    put(toString(".3",nIP1Radius[nIP1Number]))
  else
    put(toString(".3",nIP2Radius[nIP2Number]))
  endIf
  // print the X,Y,Z components of the corresponding robot Interaction Point
  // put the display for trsf values relative to the selected IP or World Frame
  //if nIPNumber==0
  if bWorldFrameView==true
    if nIPNumber==0
      LtrDisplay=fIPoriginal.trsf*fIP1.trsf*pIP1Point[nIP1Number].trsf
    else
      LtrDisplay=fIPoriginal.trsf*fIP2.trsf*pIP2Point[nIP2Number].trsf
    endIf
  else
    if nIPNumber==0
      LtrDisplay=pIP1Point[nIP1Number].trsf
    else
      LtrDisplay=pIP2Point[nIP2Number].trsf
    endIf
  endIf
  gotoxy(7,8)
  put(toString(".3",LtrDisplay.x))
  gotoxy(18,8)
  put(toString(".3",LtrDisplay.y))
  gotoxy(30,8)
  put(toString(".3",LtrDisplay.z))
  gotoxy(7,9)
  put(toString(".3",LtrDisplay.rx))
  gotoxy(18,9)
  put(toString(".3",LtrDisplay.ry))
  gotoxy(30,9)
  put(toString(".3",LtrDisplay.rz))
  // Wait indefinitely for a function button press
  LbKey=false
  getKey()
  do
    nKey=getKey()
    switch nKey
      // ESC character always ABORTS AND/OR RETURNS
      case 255
        LbKey=true
      break
      case 271,272,273,274,275,276,277,278
        LbKey=true
      break
    endSwitch
    //
    delay(0)
  until (LbKey==true)
end

--- displayMessage3.pgx ---
program displayMessage3(num nTitle (dimensions=1), num& nKey[] (dimensions=1), num XnDeltaRX (dimensions=1), num XnDeltaRY (dimensions=1), num XnDeltaRZ (dimensions=1))
  local bool LbKey
  local num LnFirst
  local num LnIndex
  local num LnQuestion
  local num LnYoffset
  local trsf LtrDisplay
begin
  //header begin
  // program displayMessage3(nTitle, nKey)
  //
  // generic pgm used for displaying complex messages and reacting to user keypad selections
  // (this program modified from pgm display2( )
  //  CUSTOMIZED SPECIFICALLY FOR TARGET FRAME / TARGET POINT ADJUSTMENT OF RX, RY, RZ
  //
  // input parms:
  //    nTitle = index of selected menu Title string in sUserPageText[ ]
  //
  //  NOTE:  the strings structure is in groups of 10 in the strings array sUserPageText[ ]
  //  Menu Page Indices are NUMBER variables
  //
  // output parms:
  //    nKey = the keypad number of the selected Function Key
  //
  // called from:  pgm mnuAdjTargetPnt()
  //
  // initial release KN
  //header end
  //
  // init local variables used as menu string text pointers
  // values are just +1 & +2 offset of nTitle pointer
  // LnYoffset used for pendant display positioning
  LnQuestion=nTitle+1
  LnFirst=nTitle+2
  LnYoffset=4
  // clear user page, and throw a title
  userPage()
  cls()
  title(sUserPageText[nTitle])
  //
  // print the Function Button Identifiers
  // at bottom of user window
  gotoxy(0,13)
  switch nSelection
    case 1
      put("Sel. Chng ---- ---- ---- ----      Ret.")
    break
    case 2,3,4
      put("Sel. ---- Inc. Dec. ---- Mov.      Ret.")
    break
  endSwitch
  //
  gotoxy(2,0)
  put("RX RY RZ adjustments applied")
  gotoxy(2,1)
  put("to current TCP location")
  gotoxy(2,3)
  put("Point data NOT SAVED on EXIT")
  //gotoxy(1,3)
  //put(sUserPageText[nTitle+3])
  //gotoxy(1,4)
  //put(sUserPageText[nTitle+4])
  gotoxy(1,5)
  put(sUserPageText[nTitle+5])
  gotoxy(1,6)
  put(sUserPageText[nTitle+6])
  gotoxy(1,7)
  put(sUserPageText[nTitle+7])
  gotoxy(1,8)
  put(sUserPageText[nTitle+8])
  gotoxy(1,9)
  put(sUserPageText[nTitle+9])
  // print the currently selected resolution
  gotoxy(18,5)
  put(toString("6.3",nResolution[nIdxResolution]))
  gotoxy(26,5)
  put("degrees")
  //
  gotoxy(18,6)
  // print adjustment value on current position's RX
  put(toString(".3",XnDeltaRX))
  // print adjustment value on current position's RY
  gotoxy(18,7)
  put(toString(".3",XnDeltaRY))
  // print adjustment value on current position's RZ
  gotoxy(18,8)
  put(toString(".3",XnDeltaRZ))
  //
  // put brackets around default selected menu item
  // nSelection is global & set in pgm mnuAdjTargetPnt()
  gotoxy(0,nSelection+LnYoffset)
  put("[>")
  gotoxy(14,nSelection+LnYoffset)
  put("<]")
  // Wait indefinitely for a function button press
  LbKey=false
  getKey()
  do
    nKey=getKey()
    switch nKey
      // ESC character always ABORTS AND/OR RETURNS
      case 255
        LbKey=true
      break
      // move selection brackets down the displayed list
      case 271
        // overwrite with blanks any previous brackets [> <]
        // offset pendant display Y location based on nSelection
        for LnIndex=(nSelection+LnYoffset) to (nSelection+LnYoffset+4)
          gotoxy(0,LnIndex)
          put("  ")
          gotoxy(14,LnIndex)
          put("  ")
        endFor
        // on F1="Sel." keypress, increment the menu item selector for bracket [> <] placement
        nSelection=nSelection+1
        if nSelection==5
          nSelection=1
        endIf
        // put [> <] around the menu item selection text
        switch nSelection
          // case=3, select "Resolution"
          case 1
            gotoxy(0,nSelection+LnYoffset)
            put("[>")
            gotoxy(14,nSelection+LnYoffset)
            put("<]")
          break
          //case=4, select "Target RX"
          case 2
            gotoxy(0,nSelection+LnYoffset)
            put("[>")
            gotoxy(14,nSelection+LnYoffset)
            put("<]")
          break
          // case=5, select "Target RY"
          case 3
            gotoxy(0,nSelection+LnYoffset)
            put("[>")
            gotoxy(14,nSelection+LnYoffset)
            put("<]")
          break
          // case=6, select "RZ"
          case 4
            gotoxy(0,nSelection+LnYoffset)
            put("[>")
            gotoxy(14,nSelection+LnYoffset)
            put("<]")
          break
          default
            popUpMsg("Bad Selection...Press OK")
          break
        endSwitch
        // print the Function Button Identifiers
        // at bottom of user window for new menu item text selection
        gotoxy(0,13)
        switch nSelection
          case 1
            put("Sel. Chng ---- ---- ---- ----      Ret.")
            //bEnableIncDec=false
          break
          case 2,3,4
            put("Sel. ---- Inc. Dec. ---- Mov.      Ret.")
          break
        endSwitch
      break
      // any other keypress, send the key num back to pgm mnuAdjTargetPnt() for changes
      case 272,273,274,276,278
        LbKey=true
      break
    endSwitch
    //
    delay(0)
  until (LbKey==true)
  //
  //done
  //
end

--- displayMessage4.pgx ---
program displayMessage4(num nTitle (dimensions=1), num& nKey[] (dimensions=1))
  local bool LbKey
  local num LnFirst
  local num LnIndex
  local num LnQuestion
  local point LpHere
  local point LpPark
begin
  //header begin
  // program displayMessage4(nTitle, nKey)
  //
  // generic pgm used for pgm checkAtPark()
  // (this program modified from pgm display( )
  //
  // input parms:
  //    nTitle = index of selected menu Title string in sUserPageText[ ]
  //
  // other parms:
  //    nQuestion = nTitle+1 = index of selected menu Question string in sUserPageText[ ]
  //    nFirst = nTitle+2 = index of the first menu Items to be displayed from sUserPageText[ ]
  //
  //  NOTE:  the strings structure is in groups of 10 in the strings array sUserPageText[ ]
  //  Menu Page Indices are NUMBER variables
  //
  // output parms:
  //    nKey = the keypad number of the selected Function Key
  //
  // called from:  various
  // initial release KN
  //header end
  //
  // init local variables used as menu string text pointers
  // values are just +1 & +2 offset of nTitle pointer
  LnQuestion=nTitle+1
  LnFirst=nTitle+2
  // clear user page, and throw a title
  userPage()
  cls()
  title(sUserPageText[nTitle])
  //
  // Print menu page Function Button Identifiers at bottom of user window
  gotoxy(0,13)
  put(sMenuBottomLine[(nTitle-1)/10])
  //
  //print QUESTION or COMMAND
  gotoxy(0,2)
  put(sUserPageText[LnQuestion])
  //
  // print 8 statements from menu string data
  for LnIndex=LnFirst to LnFirst+7
    gotoxy(1,LnIndex-LnFirst+3)
    put("(F")
    put(toString("",LnIndex-LnFirst+1))
    put(") ")
    put(sUserPageText[LnIndex])
  endFor
  //
  // test current TCP location & print the Arm Park Status
  gotoxy(0,0)
  LpHere=here(tSensorTool,world)
  LpPark=jointToPoint(tSensorTool,world,jPark)
  if (distance(LpHere,LpPark)>nParkTolerance)
    put(" Arm Park Status:  NOT PARKED! ")
  else
    put(" Arm Park Status:  PARKED & READY  ")
  endIf
  // Wait indefinitely for a function button press
  LbKey=false
  getKey()
  do
    nKey=getKey()
    switch nKey
      // ESC character always ABORTS AND/OR RETURNS
      case 255
        LbKey=true
      break
      // Function Button value returned for selected action
      case 271,272,273,274,275,276,277,278
        LbKey=true
      break
    endSwitch
    //
    delay(0)
  until (LbKey==true)
end

--- displayMessage5.pgx ---
program displayMessage5(num nTitle (dimensions=1), num& nKey[] (dimensions=1))
  local bool LbKey
  local num LnFirst
  local num LnIndex
  local num LnQuestion
begin
  //header begin
  // program displayMessage5(nTitle, nKey)
  //
  // (this program modified from pgm display( )
  // this program used specifically for pgm mnuEnterTCPVals() because of added text displayed on UserPage()
  //
  // input parms:
  //    nTitle = index of selected menu Title string in sUserPageText[ ]
  //
  // other parms:
  //    nQuestion = nTitle+1 = index of selected menu Question string in sUserPageText[ ]
  //    nFirst = nTitle+2 = index of the first menu Items to be displayed from sUserPageText[ ]
  //
  //  NOTE:  the strings structure is in groups of 10 in the strings array sUserPageText[ ]
  //  Menu Page Indices are NUMBER variables
  //
  // output parms:
  //    nKey = the keypad number of the selected Function Key
  //
  // called from:  various
  // Added for Release 2:  KN
  //
  //header end
  //
  // init local variables used as menu string text pointers
  // values are just +1 & +2 offset of nTitle pointer
  LnQuestion=nTitle+1
  LnFirst=nTitle+2
  // clear user page, and throw a title
  userPage()
  cls()
  title(sUserPageText[nTitle])
  //
  // Print menu page Function Button Identifiers at bottom of user window
  gotoxy(0,13)
  put(sMenuBottomLine[(nTitle-1)/10])
  //
  //print QUESTION or COMMAND
  gotoxy(0,2)
  put(sUserPageText[LnQuestion])
  //
  // print 8 statements from menu string data
  for LnIndex=LnFirst to LnFirst+7
    gotoxy(0,LnIndex-LnFirst+3)
    put(sUserPageText[LnIndex])
  endFor
  //
  // populate the UserPage() with {X, Y, Z, RX, RY, RZ} values of tSensorTool TCP
  gotoxy(12,3)
  put(toString(".1",tSensorTool.trsf.x))
  gotoxy(12,4)
  put(toString(".1",tSensorTool.trsf.y))
  gotoxy(12,5)
  put(toString(".1",tSensorTool.trsf.z))
  gotoxy(12,6)
  put(toString(".1",tSensorTool.trsf.rx))
  gotoxy(12,7)
  put(toString(".1",tSensorTool.trsf.ry))
  gotoxy(12,8)
  put(toString(".1",tSensorTool.trsf.rz))
  // Wait indefinitely for a function button press
  LbKey=false
  getKey()
  do
    nKey=getKey()
    switch nKey
      // ESC key always ABORTS AND / OR RETURNS
      case 255
        LbKey=true
      break
      // Function Button value returned for selected action
      case 271,272,273,274,275,276,277,278
        LbKey=true
      break
    endSwitch
    //
    delay(0)
  until (LbKey==true)
end

--- displayMessage6.pgx ---
program displayMessage6(num nTitle (dimensions=1), num& nKey[] (dimensions=1))
  local bool LbKey
  local num LnFirst
  local num LnIndex
  local num LnQuestion
begin
  //header begin
  // program displayMessage6(nTitle, nKey)
  //
  // generic pgm used for displaying complex messages and reacting to user keypad selections
  // (this program modified from pgm display( )
  // (this pgm specifically for use with pgm mnuTeachIP()
  //
  // input parms:
  //    nTitle = index of selected menu Title string in sUserPageText[ ]
  //
  // other parms:
  //    nQuestion = nTitle+1 = index of selected menu Question string in sUserPageText[ ]
  //    nFirst = nTitle+2 = index of the first menu Items to be displayed from sUserPageText[ ]
  //
  //  NOTE:  the strings structure is in groups of 10 in the strings array sUserPageText[ ]
  //  Menu Page Indices are NUMBER variables
  //
  // output parms:
  //    nKey = the keypad number of the selected Function Key
  //
  // called from:  various
  // initial release KN
  //header end
  //
  // init local variables used as menu string text pointers
  // values are just +1 & +2 offset of nTitle pointer
  LnQuestion=nTitle+1
  LnFirst=nTitle+2
  // clear user page, and throw a title
  userPage()
  cls()
  title(sUserPageText[nTitle])
  //
  // Print menu page Function Button Identifiers at bottom of user window
  gotoxy(0,13)
  put(sMenuBottomLine[(nTitle-1)/10])
  //
  //print QUESTION or COMMAND
  gotoxy(0,2)
  put(sUserPageText[LnQuestion])
  //
  // print 8 statements from menu string data
  for LnIndex=LnFirst to LnFirst+7
    gotoxy(0,LnIndex-LnFirst+3)
    put(sUserPageText[LnIndex])
  endFor
  //
  // print the TargetChoice variable for Frame Teach
  gotoxy(0,0)
  if nIPNumber==-1
    put("ACTIVE IP = Original hutch IP")
  else
    put("ACTIVE IP = "+sTargetChoice[nIPNumber])
  endIf



  // Wait indefinitely for a function button press
  LbKey=false
  getKey()
  do
    nKey=getKey()
    switch nKey
      // ESC key always ABORTS AND / OR RETURNS
      case 255
        LbKey=true
      break
      // Function Button value returned for selected action
      case 271,272,273,274,275,276,277,278
        LbKey=true
      break
    endSwitch
    //
    delay(0)
  until (LbKey==true)
end

--- displayMessage7.pgx ---
program displayMessage7(num nTitle (dimensions=1), num& nKey[] (dimensions=1))
  local bool LbKey
  local num LnFirst
  local num LnIndex
  local num LnQuestion
begin
  //header begin
  // program displayMessage7(nTitle, nKey)
  //
  // (this program modified from pgm displayMessage5( )
  // this program used specifically for pgm mnuEnterIPVals() because of added text displayed on UserPage()
  //
  // input parms:
  //    nTitle = index of selected menu Title string in sUserPageText[ ]
  //
  // other parms:
  //    nQuestion = nTitle+1 = index of selected menu Question string in sUserPageText[ ]
  //    nFirst = nTitle+2 = index of the first menu Items to be displayed from sUserPageText[ ]
  //
  //  NOTE:  the strings structure is in groups of 10 in the strings array sUserPageText[ ]
  //  Menu Page Indices are NUMBER variables
  //
  // output parms:
  //    nKey = the keypad number of the selected Function Key
  //
  // called from:  various
  // Added for Release 2:  KN
  //
  //header end
  //
  // init local variables used as menu string text pointers
  // values are just +1 & +2 offset of nTitle pointer
  LnQuestion=nTitle+1
  LnFirst=nTitle+2
  // clear user page, and throw a title
  userPage()
  cls()
  title(sUserPageText[nTitle])
  //
  // Print menu page Function Button Identifiers at bottom of user window
  gotoxy(0,13)
  put(sMenuBottomLine[(nTitle-1)/10])
  //
  //print QUESTION or COMMAND
  gotoxy(0,2)
  put(sUserPageText[LnQuestion])
  //
  // print 8 statements from menu string data
  for LnIndex=LnFirst to LnFirst+7
    gotoxy(0,LnIndex-LnFirst+3)
    put(sUserPageText[LnIndex])
  endFor
  //
  // populate the UserPage() with {X, Y, Z, RX, RY, RZ} values of the selected Interaction Point
  if nIPNumber==-1
    gotoxy(12,3)
    put(toString(".1",fIPoriginal.trsf.x))
    gotoxy(12,4)
    put(toString(".1",fIPoriginal.trsf.y))
    gotoxy(12,5)
    put(toString(".1",fIPoriginal.trsf.z))
    gotoxy(12,6)
    put(toString(".1",fIPoriginal.trsf.rx))
    gotoxy(12,7)
    put(toString(".1",fIPoriginal.trsf.ry))
    gotoxy(12,8)
    put(toString(".1",fIPoriginal.trsf.rz))
  elseIf nIPNumber==0
    gotoxy(12,3)
    put(toString(".1",fIP1.trsf.x))
    gotoxy(12,4)
    put(toString(".1",fIP1.trsf.y))
    gotoxy(12,5)
    put(toString(".1",fIP1.trsf.z))
    gotoxy(12,6)
    put(toString(".1",fIP1.trsf.rx))
    gotoxy(12,7)
    put(toString(".1",fIP1.trsf.ry))
    gotoxy(12,8)
    put(toString(".1",fIP1.trsf.rz))
  else
    gotoxy(12,3)
    put(toString(".1",fIP2.trsf.x))
    gotoxy(12,4)
    put(toString(".1",fIP2.trsf.y))
    gotoxy(12,5)
    put(toString(".1",fIP2.trsf.z))
    gotoxy(12,6)
    put(toString(".1",fIP2.trsf.rx))
    gotoxy(12,7)
    put(toString(".1",fIP2.trsf.ry))
    gotoxy(12,8)
    put(toString(".1",fIP2.trsf.rz))
  endIf
  // Wait indefinitely for a function button press
  LbKey=false
  getKey()
  do
    nKey=getKey()
    switch nKey
      // ESC key always ABORTS AND / OR RETURNS
      case 255
        LbKey=true
      break
      // Function Button value returned for selected action
      case 271,272,273,274,275,276,277,278
        LbKey=true
      break
    endSwitch
    //
    delay(0)
  until (LbKey==true)
end

--- displayMessage8.pgx ---
program displayMessage8(num nTitle (dimensions=1), num& nKey[] (dimensions=1))
  local bool LbKey
  local num LnFirst
  local num LnIndex
  local num LnQuestion
  local point LpCurrentLoc
begin
  //header begin
  // program displayMessage8(nTitle, nKey)
  //
  // generic pgm used for displaying complex messages and reacting to user keypad selections
  // (this program modified from pgm displayMessage( )
  // This program uses specifically for pgm mnuGetTCP()
  // Displays the values of TCP location of tSensorTool relative to selected nIPNumber Interaction Point frame.
  //
  // input parms:
  //    nTitle = index of selected menu Title string in sUserPageText[ ]
  //
  // other parms:
  //    nQuestion = nTitle+1 = index of selected menu Question string in sUserPageText[ ]
  //    nFirst = nTitle+2 = index of the first menu Items to be displayed from sUserPageText[ ]
  //
  //  NOTE:  the strings structure is in groups of 10 in the strings array sUserPageText[ ]
  //  Menu Page Indices are NUMBER variables
  //
  // output parms:
  //    nKey = the keypad number of the selected Function Key
  //
  // called from:  various
  //
  // Release History:
  //  This pgm released as part of SLAC RX130L robot control program Revision 3
  //  per Blue Technik proposal K01c, Work Request K01-1
  //
  //header end
  //
  // init local variables used as menu string text pointers
  // values are offset of nTitle pointer
  LnFirst=nTitle+1
  // clear user page, and throw a title
  userPage()
  cls()
  title(sUserPageText[nTitle])
  //
  // Print menu page Function Button Identifiers at bottom of user window
  gotoxy(0,13)
  put(sMenuBottomLine[(nTitle-1)/10])
  //
  // print 8 statements from menu string data
  for LnIndex=LnFirst to LnFirst+7
    gotoxy(0,LnIndex)
    put(sUserPageText[LnIndex])
  endFor
  //
  // Populate teh User Page with current IP selection & the current IP:TCP.trsf values
  if nIPNumber==0
    LpCurrentLoc=here(tSensorTool,fIP1)
  else
    LpCurrentLoc=here(tSensorTool,fIP2)
  endIf
  //
  gotoxy(14,3)
  put(toString(".0",nIPNumber))
  gotoxy(14,4)
  put(toString("5.2",LpCurrentLoc.trsf.x))
  gotoxy(14,5)
  put(toString("5.2",LpCurrentLoc.trsf.y))
  gotoxy(14,6)
  put(toString("5.2",LpCurrentLoc.trsf.z))
  gotoxy(14,7)
  put(toString("5.2",LpCurrentLoc.trsf.rx))
  gotoxy(14,8)
  put(toString("5.2",LpCurrentLoc.trsf.ry))
  gotoxy(14,9)
  put(toString("5.2",LpCurrentLoc.trsf.rz))
  //
  // Wait indefinitely for a function button press
  LbKey=false
  getKey()
  do
    nKey=getKey()
    switch nKey
      // ESC key always ABORTS AND / OR RETURNS
      case 255
        LbKey=true
      break
      // Function Button value returned for selected action
      case 271,278
        LbKey=true
      break
    endSwitch
    //
    delay(0)
  until (LbKey==true)
end

--- displayMessage9.pgx ---
program displayMessage9(num nTitle (dimensions=1), num& nKey[] (dimensions=1))
  local bool LbKey
  local num LnFirst
  local num LnIndex
  local num LnQuestion
begin
  //header begin
  // program displayMessage9(nTitle, nKey)
  //
  // generic pgm used for displaying complex messages and reacting to user keypad selections
  // used for testing if bSimulateESTOP is active
  //
  // input parms:
  //    nTitle = index of selected menu Title string in sUserPageText[ ]
  //
  // other parms:
  //    nQuestion = nTitle+1 = index of selected menu Question string in sUserPageText[ ]
  //    nFirst = nTitle+2 = index of the first menu Items to be displayed from sUserPageText[ ]
  //
  //  NOTE:  the strings structure is in groups of 10 in the strings array sUserPageText[ ]
  //  Menu Page Indices are NUMBER variables
  //
  // output parms:
  //    nKey = the keypad number of the selected Function Key
  //
  // called from:  mnuTestSimESTOP()
  // initial release KN
  //header end
  //
  // init local variables used as menu string text pointers
  // values are just +1 & +2 offset of nTitle pointer
  LnQuestion=nTitle+1
  LnFirst=nTitle+2
  // clear user page, and throw a title
  userPage()
  cls()
  title(sUserPageText[nTitle])
  //
  // Print menu page Function Button Identifiers at bottom of user window
  gotoxy(0,13)
  put(sMenuBottomLine[(nTitle-1)/10])
  //
  //print QUESTION or COMMAND
  gotoxy(0,2)
  put(sUserPageText[LnQuestion])
  //
  // print 8 statements from menu string data
  for LnIndex=LnFirst to LnFirst+7
    gotoxy(0,LnIndex-LnFirst+3)
    put(sUserPageText[LnIndex])
  endFor
  //
  LbKey=false
  getKey()
  do
    nKey=getKey()
    switch nKey
      // Function Button value returned for selected action
      case 271,278
        LbKey=true
      break
    endSwitch
    //
    delay(0)
  until (LbKey==true)
end

--- initialize.pgx ---
public program initialize()
  local num LnIndex
begin
  // header begin
  //
  // Program initialize( )
  // This program initializes variables
  //
  // incoming parms:  none
  // outgoing parms:  none
  // called from:  pgm main()
  //
  // initial release KN
  //
  //header end
  //
  //==== numbers =================
  nNumberCube=0
  nNumberCylinder=0
  nNumberSphere=0
  nDistXCube=0
  nDistYCube=0
  nDistZCube=0
  nDistZCylinder=0
  nRadiusCylinder=0
  nRadiusSphere=0
  nMaxLoginTries=3
  nParkTolerance=50
  nAccSlow=20
  nAccMedium=40
  nAccFast=60
  nVelSlow=20
  nVelMedium=40
  nVelFast=60
  nZoneWatchTol=25
  nAdjPntMoveTol=25
  nParkTolerance=50
  nRemoteTimeout=30
  nMaxVelo=100
  nMaxRVelo=20
  nMaxAccel=50
  nMaxDist=1000
  sNumConv=".3"
  //
  //==== location points =========
  pIP1NullPoint.trsf={0,0,0,0,0,0}
  pIP2NullPoint.trsf={0,0,0,0,0,0}
  pMoveIP1Target.trsf={0,0,0,0,0,0}
  pMoveIP2Target.trsf={0,0,0,0,0,0}
  pNullPosition.trsf={0,0,0,0,0,0}
  //
  //==== frames ===================
  //
  //==== booleans =================
  bStopAllMonitor=true
  bEnableMonitor=false
  bRemControlON=false
  bSimulateESTOP=true
  bMoveLinear=true
  //
  //==== input signals ============
  //
  //==== output signals ===========
  //
  //==== strings ==================
  sIOCUserName="CS8LOGIN"
  sIOCPassword="USERPASSWORD"
  //
  //==== comm & serial port =======
  sioLink(sioIOCclient,io:IOC)
  //
  //==== tool definitions =========
  //tSensorTool.trsf=tNULLTOOL.trsf*{0,0,300,0,0,0}*{0,0,0,0,90,0}*{0,0,0,0,0,90}
  //tRefPointer.trsf={0,0,200,0,0,0}
  //
  //==== motion descriptor ========t
  mDefault.accel=mDefault.decel=20
  mDefault.vel=20
  mGlobalSpeed=mDefault
  // done
end

--- initializeRobot.pgx ---
program initializeRobot()
  local bool LbArmPowerOn
  local bool LbESTOPActive
  local num LnKey
  local num nKey
begin
  //header begin
  // PROGRAM initializeRobot()
  //
  // checks for necessary conditions to be met before any robot movement under automatic control
  //    ESTOP is not active
  //    Arm Power = ON
  //    Arm is Calibrated
  //
  // incoming parms:  none
  // outgoing parms:  none
  // called from:  pgm mnuUtilityMenu()
  //               pgm movTargetPoint()
  //
  //  initial release KN
  //header end
  //
  // clear motion stack of all movement commands
  stopMove()
  resetMotion()
  //
  userPage()
  cls()
  //
  // verify ESTOP is inactive
  title(" ESTOP CHECK ")
  putln("Check ESTOP status...")
  if (esStatus()==2)
    LbESTOPActive=true
    userPage()
    cls()
    title(" RESET ESTOP ")
    gotoxy(0,4)
    putln("WAITING:  Reset ESTOP")
    wait(esStatus()==0)
  else
    putln("OK")
  endIf
  //
  // Have user put system into MANUAL MODE
  cls()
  title(" MANUAL MODE CHECK ")
  putln("Check Working Mode...")
  if (workingMode()!=1)
    userPage()
    cls()
    title(" SELECT MANUAL MODE ")
    gotoxy(0,4)
    putln("WAITING:  Select MANUAL MODE")
    wait(workingMode()==1)
  else
    putln("OK, Manual Mode")
  endIf
  //
  // Have user verify Arm Power is ON.  Use pgm display() for menu control.
  cls()
  title(" ARM POWER CHECK ")
  putln("Check Arm Power...")
  //
  // Have user verify arm is calibrated. Use pgm display() for menu control.
  // If not calibrated, user must abort & stop application, calibrate, then restart application.
  // This menu allows user to return to previous menu.
  cls()
  title(" ARM CALIBRATION CHECK ")
  putln("Checking Arm Calibration...")
  if (isCalibrated()==false)
    cls()
    gotoxy(0,4)
    putln("WARNING!  ARM REQUIRES CALIBRATION")
    gotoxy(0,6)
    putln("Press any key to shut down...")
    do
      LnKey=getKey()
      delay(0.25)
    until LnKey!=-1
    cls()
    call stop()
  else
    putln("OK, Arm is calibrated")
  endIf
  //
  // done
end

--- iocWriteBack.pgx ---
program iocWriteBack(string XsResponse (dimensions=1))
begin
  //
  //header begin
  // PROGRAM iocWriteBack()
  //
  // pgm writes text via TCP/IP to IOC client socket on CS8
  //
  // input parms:
  //    XsResponse = string passed from calling program
  //
  // output parms:
  //    none
  //
  // called from:  iocCmdHandler()
  //
  // initial release:  KN
  // Release 2:  KN
  //  changed functionality from CS8 host to CS8 client
  //  updated documentation
  //header end
  //
  sioIOCclient=XsResponse
end

--- makePntAZELRA.pgx ---
program makePntAZELRA(num XnIPNumber (dimensions=1), num XnTPNumber (dimensions=1))
begin
  //header begin
  // PROGRAM makePntAZELRA()
  //
  // transforms all Azimuth-Elevation-Radius input data to
  // Cartesian {X, Y, Z, rX, rY, rZ} points
  // done globally, works on single point only
  //
  // incoming parms:
  //    XnIPNumber = currently selected Interaction Point Number, either 0=IP1 or 1=IP2
  //    XnTPNumber = currently selected Target Point Number, range=0-19
  // outgoing parms:  none
  // called from:  pgm mnuSetTargetPts()
  //
  // NEW DEFINITION TO MATCH SLAC SPECIFICATION MATH DESCRIPTION
  //    For fIPn aligned so that
  //      fIPn_+Zaxis in direction of beam travel and parallel to RX160L World_+Yaxis
  //      fIPn_+Xaxis parallel to pointing to IOC Hutch entrance doors & parallel to RX160L World_+Xaxis
  //      fIPn_+Yaxis pointing to ceiling and parallel to RX160L World_-Zaxis
  //          NOTE:  these statements are valid for BOTH fIP1 & fIP2 since the robot is on translating base
  //                 does not have to reach "over" to another fIPn
  //    Therefore
  //      Azimuth = rotation about fIPn_Yaxis
  //      Elevation = rotation about fIPn_Z'axis
  //      Radius = translation along fIPn_X'axis
  //
  //  initial release KN
  //  updated @SLAC 17feb2010 KN
  //header end
  //
  // updates for IP1 Target Points
  if XnIPNumber==0
    //
    // new definitions to match SLAC spec math
    pIP1Point[XnTPNumber].trsf={0,0,0,0,0,0}
    // Add AZ component:  rotate about fIPn_+Yaxis
    pIP1Point[XnTPNumber].trsf=pIP1Point[XnTPNumber].trsf*{0,0,0,0,nIP1Azimuth[XnTPNumber],0}
    // Add EL component:  rotate about fIPn_+Z'axis
    pIP1Point[XnTPNumber].trsf=pIP1Point[XnTPNumber].trsf*{0,0,0,-nIP1Elevation[XnTPNumber],0,0}
    // Add RA component:  translate along fIPn+X'axis
    pIP1Point[XnTPNumber].trsf=pIP1Point[XnTPNumber].trsf*{0,0,nIP1Radius[XnTPNumber],0,0,0}
    // now transform the point so that +Zaxis points back to fIPn
    pIP1Point[XnTPNumber].trsf=pIP1Point[XnTPNumber].trsf*{0,0,0,0,-180,0}
    pIP1Point[XnTPNumber].config={sfree,efree,wfree}
    //
  endIf
  //
  // updates for IP2 Target Points
  if XnIPNumber==1
    //
    // new definitions to match SLAC spec math (as above)
    pIP2Point[XnTPNumber].trsf={0,0,0,0,0,0}
    pIP2Point[XnTPNumber].trsf=pIP2Point[XnTPNumber].trsf*{0,0,0,0,nIP2Azimuth[XnTPNumber],0}
    pIP2Point[XnTPNumber].trsf=pIP2Point[XnTPNumber].trsf*{0,0,0,-nIP2Elevation[XnTPNumber],0,0}
    pIP2Point[XnTPNumber].trsf=pIP2Point[XnTPNumber].trsf*{0,0,nIP2Radius[XnTPNumber],0,0,0}
    pIP2Point[XnTPNumber].trsf=pIP2Point[XnTPNumber].trsf*{0,0,0,0,-180,0}
    pIP2Point[XnTPNumber].config={sfree,efree,wfree}
    //
  endIf
  // done
end

--- mnuAdjTargetPnt.pgx ---
public program mnuAdjTargetPnt()
  local bool LbBackup
  local bool LbMoveOutOfTol
  local num LnDeltaRX
  local num LnDeltaRY
  local num LnDeltaRZ
  local num LnDistance
  local point LpHere
  local point LpTargetPoint
  local point LpTempAdjPoint
  local num nKey
begin
  //header begin
  // PROGRAM mnuAdjTargetPnt()
  //
  // runs the menu to query user for all info needed to adjust RX RY RZ of Target Points
  // adjusts, but does not save the new point definition because the point would then not
  // be consistent with the AZ EL RA root definition of the point location.
  //
  // incoming parms:  none
  //
  // outgoing parms:  none
  // called from:  pgm mnuMoveTargPnt()
  //
  //  initial release KN
  //header end
  //
  // start continuous loop, end by menu command or teach pendant command
  // on user command, jump to other subroutines for action
  //
  // init booleans for menu control
  LbBackup=false
  nSelection=1
  nIdxResolution=0
  LnDeltaRX=0
  LnDeltaRY=0
  LnDeltaRZ=0
  LpTempAdjPoint=here(tSensorTool,world)
  //
  // test if at currently selected Target Point before Adjustment Move
  // Deny adjustment if not within nAdjPntMoveTol and return
  LpHere=here(tSensorTool,world)
  if nIPNumber==0
    LpTargetPoint=pIP1Point[nIP1Number]
  else
    LpTargetPoint=pIP2Point[nIP2Number]
  endIf
  LnDistance=abs(distance(LpHere,LpTargetPoint))
  if LnDistance>nAdjPntMoveTol
    popUpMsg("ADJUSTMENT DENIED:  Sensor Tool TCP not at selected Target Point...Press OK")
  else
    do
      //nIdxAdjTargetPt=291
      call displayMessage3(nIdxAdjTargetPt,nKey,LnDeltaRX,LnDeltaRY,LnDeltaRZ)
      // verify selection
      switch nKey
        // ESC aborts/returns immediately, no save
        case 255
          return
        break
        // menu = Adj Target Point, F2 to Change (increment) the values of
        // Resolution ONLY
        case 272
          switch nSelection
            // cycle through the available resolutions
            case 1
              nIdxResolution=nIdxResolution+1
              if nIdxResolution==4
                nIdxResolution=0
              endIf
            break
          endSwitch
        break
        // menu=Adj Target Pnts, F3 increments by nResolution RX, RY, RZ as selected by nSelection
        case 273
          switch nSelection
            // select & increment RX
            case 2
              LnDeltaRX=LnDeltaRX+nResolution[nIdxResolution]
            break
            // select & increment RY
            case 3
              LnDeltaRY=LnDeltaRY+nResolution[nIdxResolution]
            break
            // select & increment RZ
            case 4
              LnDeltaRZ=LnDeltaRZ+nResolution[nIdxResolution]
            break
          endSwitch
        break
        //  menu = Adj Targ Pnts, F4 to Decrement by resolution
        case 274
          switch nSelection
            // select & decrement RX
            case 2
              LnDeltaRX=LnDeltaRX-nResolution[nIdxResolution]
            break
            // select & decrement RY
            case 3
              LnDeltaRY=LnDeltaRY-nResolution[nIdxResolution]
            break
            // select & decrement RZ
            case 4
              LnDeltaRZ=LnDeltaRZ-nResolution[nIdxResolution]
            break
          endSwitch
        break
        // menu = AdjTarget Point
        // F6 = Command a move to adjusted value determined by selection
        case 276
          // no Zone Monitoring done during Adjustment moves
          // no checking of valid moves
          cls()
          title(" ADJUST RX/RY/RZ MOVE ")
          gotoxy(0,2)
          putln("WAITING:  Press MOVE/HOLD Button")
          putln("          to move to RX/RY/RZ Adj Point")
          LpTempAdjPoint.trsf=LpTempAdjPoint.trsf*{0,0,0,LnDeltaRX,LnDeltaRY,LnDeltaRZ}
          movel(LpTempAdjPoint,tSensorTool,mGlobalSpeed)
          waitEndMove()
          cls()
          popUpMsg("Target Point Adjustment Move COMPLETED...Press OK")
        break
        // menu = Adjust Interaction Point Target Point, F7 to SAVE Adjusted Point Data, no return
        //  menu = Adj Targ Pnts, F8 returns with no save
        case 278
          LbBackup=true
        break
        // Any other key press
        default
          cls()
          popUpMsg("BAD SELECTION...press OK")
        break
      endSwitch
    until (false or (LbBackup==true))
    //
  endIf
  // done
end

--- mnuEnterIPVals.pgx ---
program mnuEnterIPVals()
  local bool LbBackup
  local num nKey
begin
  //
  //header begin
  //
  //  pgm mnuEnterIPVals()
  // this program allows user to set global Interaction Point values
  //
  //  incoming parms: none
  //  outgoing parms: none
  //
  //  called from mnuTeachIP()
  //
  //  Added for Release 2: KN
  //
  //header end
  //
  // set up display
  LbBackup=false
  do
    // nIdxEnterIP=341
    call displayMessage7(nIdxEnterIP,nKey)
    // verify selection
    switch nKey
      // ESC key aborts immediately
      case 255
        return
      break
      // menu = Direct Entry TCP values, F1 button = IP-X value
      case 271
        gotoxy(18,3)
        if nIPNumber==-1
          get(fIPoriginal.trsf.x)
        elseIf nIPNumber==0
          get(fIP1.trsf.x)
        else
          get(fIP2.trsf.x)
        endIf
      break
      // menu = Direct Entry TCP values,  F2 Button = IP-Y value
      case 272
        gotoxy(18,4)
        if nIPNumber==-1
          get(fIPoriginal.trsf.y)
        elseIf nIPNumber==0
          get(fIP1.trsf.y)
        else
          get(fIP2.trsf.y)
        endIf
      break
      // menu = Direct Entry TCP Values,  F3 Button = IP-Z value
      case 273
        gotoxy(18,5)
        if nIPNumber==-1
          get(fIPoriginal.trsf.z)
        elseIf nIPNumber==0
          get(fIP1.trsf.z)
        else
          get(fIP2.trsf.z)
        endIf
      break
      // menu = Direct Entry TCP values, F4 Button = IP-RX value
      case 274
        gotoxy(18,6)
        if nIPNumber==-1
          get(fIPoriginal.trsf.rx)
        elseIf nIPNumber==0
          get(fIP1.trsf.rx)
        else
          get(fIP2.trsf.rx)
        endIf
      break
      // menu = Direct Entry TCP Values, F5 Button = IP-RY value
      case 275
        gotoxy(18,7)
        if nIPNumber==-1
          get(fIPoriginal.trsf.ry)
        elseIf nIPNumber==0
          get(fIP1.trsf.ry)
        else
          get(fIP2.trsf.ry)
        endIf
      break
      // menu = Direct Entry TCP Values, F6 Button = IP-RZ value
      case 276
        gotoxy(18,8)
        if nIPNumber==-1
          get(fIPoriginal.trsf.rz)
        elseIf nIPNumber==0
          get(fIP1.trsf.rz)
        else
          get(fIP2.trsf.rz)
        endIf
      break
      // menu = Main Menu:  F8 Button, Save updated TCP values & return to pgm mnuTeachIP()
      case 278
        LbBackup=true
        libSave()
      break
      // ALL OTHER CHOICES
      default
        popUpMsg("EnterIPVals:  BAD SELECTION...Press OK")
      break
    endSwitch
  until (false or (LbBackup==true))
end

--- mnuEnterTCPVals.pgx ---
program mnuEnterTCPVals()
  local bool LbBackup
  local num nKey
begin
  //
  //header begin
  //
  //  pgm mnuEnterTCPVals()
  // this program allows user to set global TCP values on tSensorTool
  //
  //  incoming parms: none
  //  outgoing parms: none
  //
  //  called from mnuTeachTCP()
  //
  //  Added for Release 2: KN
  //
  //header end
  //
  // set up display
  LbBackup=false
  do
    // nIdxEnterTCP=321
    call displayMessage5(nIdxEnterTCP,nKey)
    // verify selection
    switch nKey
      // ESC key aborts immediately
      case 255
        return
      break
      // menu = Direct Entry TCP values, F1 button = TCP-X value
      case 271
        gotoxy(18,3)
        get(tSensorTool.trsf.x)
      break
      // menu = Direct Entry TCP values,  F2 Button = TCP-Y value
      case 272
        gotoxy(18,4)
        get(tSensorTool.trsf.y)
      break
      // menu = Direct Entry TCP Values,  F3 Button = TCP-Z value
      case 273
        gotoxy(18,5)
        get(tSensorTool.trsf.z)
      break
      // menu = Direct Entry TCP values, F4 Button = TCP-RX value
      case 274
        gotoxy(18,6)
        get(tSensorTool.trsf.rx)
      break
      // menu = Direct Entry TCP Values, F5 Button = TCP-RY value
      case 275
        gotoxy(18,7)
        get(tSensorTool.trsf.ry)
      break
      // menu = Direct Entry TCP Values, F6 Button = TCP-RZ value
      case 276
        gotoxy(18,8)
        get(tSensorTool.trsf.rz)
      break
      // menu = Main Menu:  F8 Button, Save updated TCP values & return to pgm mnuTeachTCP()
      case 278
        LbBackup=true
        libSave()
      break
      // ALL OTHER CHOICES
      default
        popUpMsg("BAD SELECTION...Press OK")
      break
    endSwitch
  until (false or (LbBackup==true))
end

--- mnuGetTCP.pgx ---
program mnuGetTCP()
  local bool LbBackup
  local num nKey
begin
  //header begin
  // PROGRAM mnuGetTCP()
  //
  // runs the menu to show current TCP values for tSensorTool at the currently selected
  // /Interaction Point frame.  Allows the user to toggle the selection of the IP Frame.
  //
  // incoming parms:  none
  // outgoing parms:  none
  // called from:  pgm mnuUtilityMenu()
  //
  //  This program is released as part of SLAC RX130L robot control code Revision 3.
  //  This is part of Blue Technik proposal K01c, Work Request K01-1.
  //header end
  //
  // start continuous loop, end by menu command or teach pendant command
  // on user command, jump to other subroutines for action
  //
  // init booleans for menu control in pgm displayMessage2()
  LbBackup=false
  //
  do
    //nIdxSetTargetPt=351
    call displayMessage8(nIdxGetTCP,nKey)
    // verify selection
    switch nKey
      // ESC key aborts, return with no save to pgm mnuTeachMenu()
      case 255
        return
      break
      // menu = Get TCP Values @ IP,
      // F1 to change Interaction Point number 0 or 1
      case 271
        nIPNumber=nIPNumber+1
        if nIPNumber==2
          nIPNumber=0
        endIf
      break
      //  menu = Get TCP Values @ IP, F8 to exit & return to pgm mnuUtilityMenu()
      case 278
        LbBackup=true
      break
      // Any other key press
      default
        cls()
        popUpMsg("BAD SELECTION...press OK")
      break
    endSwitch
  until (false or (LbBackup==true))
  //
  // done
end

--- mnuGlobalSpeed.pgx ---
program mnuGlobalSpeed()
  local bool LbBackup
  local num nKey
begin
  //
  //header begin
  //
  //  pgm mnuGlobalSpeed()
  // this program allows user to set global motion descriptor values from pre-defined set
  //
  //  incoming parms: none
  //  outgoing parms: none
  //
  //  called from mnuUtility()
  //
  //  initial release KN
  //
  //header end
  //
  // set up display
  LbBackup=false
  do
    // nIdxSetSpeeds=181
    call display(nIdxSetSpeeds,nKey)
    // verify selection
    switch nKey
      // ESC key aborts immediately
      case 255
        return
      break
      // menu = Set Global Speed Parms:  F1 Button, set Slow speed
      case 271
        mGlobalSpeed.vel=nVelSlow
        LbBackup=true
        popUpMsg("Global Velocity set to SLOW...Press OK")
      break
      // menu = Set Global Speed Parms:  F2 Button, set Medium Speed
      case 272
        mGlobalSpeed.vel=nVelMedium
        LbBackup=true
        popUpMsg("Global Velocity set to MEDIUM...Press OK")
      break
      // menu = Set Global Speed Parms:  F3 Button, set Fast Speed
      case 273
        mGlobalSpeed.vel=nVelFast
        LbBackup=true
        popUpMsg("Global Velocity set to FAST...Press OK")
      break
      // menu = Set Global Speed Parms, F5 Button = set Slow Accels
      case 275
        mGlobalSpeed.accel=mGlobalSpeed.decel=nAccSlow
        LbBackup=true
        popUpMsg("Global Accel/decel set to SLOW...Press OK")
      break
      // menu = Set Global Speed Parms, F6 Button = set Medium Accels
      case 276
        mGlobalSpeed.accel=mGlobalSpeed.decel=nAccMedium
        LbBackup=true
        popUpMsg("Global Accel/Decel set to MEDIUM...Press OK")
      break
      // menu = Set Global Speed Parms, F7 Button = set Fast Accels
      case 277
        mGlobalSpeed.accel=mGlobalSpeed.decel=nAccFast
        LbBackup=true
        popUpMsg("Global Accel/Decel set to FAST...Press OK")
      break
      // menu = Main Menu:  F8 Button, End Application & Exit
      case 278
        LbBackup=true
      break
      // ALL OTHER CHOICES
      default
        popUpMsg("BAD SELECTION...Press OK")
      break
    endSwitch
  until (false or (LbBackup==true))
end

--- mnuMotionMenu.pgx ---
program mnuMotionMenu()
  local bool LbBackup
  local num nKey
begin
  //header begin
  // PROGRAM mnuMotionMenu()
  //
  // runs the menu to select various MOTION functions
  //
  // incoming parms:  none
  // outgoing parms:  none
  // called from:  pgm main()
  //
  //  initial release KN
  //  Release 3:  added F3 Button call to pgm <something>
  //  /per Blue Technik quote K01c, Work Request K01-1
  //header end
  //
  // start continuous loop, end by menu command or teach pendant command
  // on user command, jump to other subroutines for action
  //
  LbBackup=false
  do
    //nIdxMotionMenu=271
    call display(nIdxMotionMenu,nKey)
    // verify selection
    switch nKey
      // ESC key aborts & returns immediately
      case 255
        return
      break
      // Motion Menu:  F1 Button, go to Target Point menu for move & adjust functions
      case 271
        call mnuMoveTargPnt()
      break
      // Motion Menu:  F4 Button, Move to PARK position
      case 274
        call movToPark()
      break
      // Motion Menu:  F6 Button, Move to PARK TOP position
      case 276
        call movToParkTop()
      break
      // F8 Button, backup to Main Menu
      case 278
        LbBackup=true
      break
      // any other key press
      default
        cls()
        popUpMsg("BAD SELECTION...Press OK")
      break
    endSwitch
  until (false or (LbBackup==true))
  // done
end

--- mnuMoveTargPnt.pgx ---
program mnuMoveTargPnt()
  local bool LbBackup
  local bool LbIsInRange
  local bool LbTestLocResult
  local joint LjHere
  local joint LjTarget
  local point LpMoveTarget
  local num nKey
begin
  //header begin
  // PROGRAM mnuMoveTargPnt()
  //
  // runs the menu to query for user to select and move to
  // Target Point
  //
  // incoming parms:  none
  // outgoing parms:  none
  // called from:  pgm mnuMotionMenu()
  //
  //  initial release KN
  //header end
  //
  // start continuous loop, end by menu command or teach pendant command
  // on user command, jump to other subroutines for action
  //
  // init booleans for menu control
  LbBackup=false
  bWorldFrameView=true
  //
  do
    //nIdxMoveTargPt=281
    call displayMessage2(nIdxMoveTargPt,nKey)
    // verify selection
    switch nKey
      // ESC key aborts & returns immediately
      case 255
        return
      break
      // Move to Target Point, F1 to change Target Frame number 1 or 2
      case 271
        nIPNumber=nIPNumber+1
        if nIPNumber==2
          nIPNumber=0
        endIf
      break
      // Move to Target Point, F2 to increment point number 0-19 in selected frame 0-1
      case 272
        if nIPNumber==0
          nIP1Number=nIP1Number+1
          if nIP1Number==20
            nIP1Number=0
          endIf
        else
          nIP2Number=nIP2Number+1
          if nIP2Number==20
            nIP2Number=0
          endIf
        endIf
      break
      // menu Move To Target Point, F5 to ADJUST RX/RY/RZ values of Target Point
      case 275
        call mnuAdjTargetPnt()
      break
      //  Move to Target Point, F6 to MOVE to currently selected IP & TP
      case 276
        // test if move to Target Point is possible
        // set up dummy loc at current location & configuration
        LjHere=jPark
        // test desired Target Point for validity
        if nIPNumber==0


          logMsg("x  "+toString(".6",tSensorTool.trsf.x))
          logMsg("y  "+toString(".6",tSensorTool.trsf.y))
          logMsg("z  "+toString(".6",tSensorTool.trsf.z))
          logMsg("rx "+toString(".6",tSensorTool.trsf.rx))
          logMsg("ry "+toString(".6",tSensorTool.trsf.ry))
          logMsg("rz "+toString(".6",tSensorTool.trsf.rz))

          logMsg("x  "+toString(".6",pIP1Point[nIP1Number].trsf.x))
          logMsg("y  "+toString(".6",pIP1Point[nIP1Number].trsf.y))
          logMsg("z  "+toString(".6",pIP1Point[nIP1Number].trsf.z))
          logMsg("rx "+toString(".6",pIP1Point[nIP1Number].trsf.rx))
          logMsg("ry "+toString(".6",pIP1Point[nIP1Number].trsf.ry))
          logMsg("rz "+toString(".6",pIP1Point[nIP1Number].trsf.rz))


          LbTestLocResult=pointToJoint(tSensorTool,LjHere,pIP1Point[nIP1Number],LjTarget)
        else
          LbTestLocResult=pointToJoint(tSensorTool,LjHere,pIP2Point[nIP2Number],LjTarget)
        endIf
        // issue error if not valid or if cannot be reached, otherwise commence move
        if LbTestLocResult==false
          LbBackup=true
          popUpMsg("IMPOSSIBLE MOVE:  Unable to reach Target Point in current arm configuration...Press OK")
          //call movTargetPoint()
        else
          LbIsInRange=isInRange(LjTarget)
          if LbIsInRange==true
            call movTargetPoint()
          else
            popUpMsg("IMPOSSIBLE MOVE:  Target Point out of reach or out of limits...Press OK")
          endIf
        endIf
      break
      // menu = Move Target Points, F7 to change displayed trsf values relative to the selected IP or World CoordSys
      // this boolean is acted upon in pgm displayMessage2()
      case 277
        if bWorldFrameView==true
          bWorldFrameView=false
        else
          bWorldFrameView=true
        endIf
      break
      //F8 to Go Back
      case 278
        LbBackup=true
      break
      // Any other key press
      default
        popUpMsg("BAD SELECTION...press OK")
      break
    endSwitch
  until (false or (LbBackup==true))
  // done
end

--- mnuMoveToPark.pgx ---
program mnuMoveToPark()
  local bool LbBackup
  local num nKey
begin
  //header begin
  // PROGRAM mnuMoveToPark()
  //
  // runs the menu to guide user to Move to PARK Location
  //
  // incoming parms:  none
  // outgoing parms:  none
  // called from:  pgm main()
  //
  //  initial release KN
  //header end
  //
  // start continuous loop, end by menu command or teach pendant command
  // on user command, jump to other subroutines for action
  //
  LbBackup=false
  do
    //nIdxMotionMenu=311
    call display(nIdxMoveToPark,nKey)
    // verify selection
    switch nKey
      // ESC key aborts & returns immediately
      case 255
        return
      break
      // menu = MoveToPark  F1 Button, Move to PARK Location
      case 271
        //        stopMove()
        //        resetMotion()
        //        // check robot condition
        //        call initializeRobot()
        //        userPage()
        //        cls()
        //        title(" MOVE TO PARK ")
        //        gotoxy(0,4)
        //        putln("WAITING:  Press MOVE/HOLD button")
        //        putln("          to move to Park...")
        //        //
        //        bEnableMonitor=true
        //        LpPark=jointToPoint(tSensorTool,world,jPark)
        //        movel(LpPark,tSensorTool,mGlobalSpeed)
        //        waitEndMove()
        //        bEnableMonitor=false
        //        popUpMsg("NOW AT PARK...Press OK")
        //        LbBackup=true
        call movToPark()
      break
      // F8 Button, backup to Main Menu
      case 278
        LbBackup=true
      break
      // any other key press
      default
        cls()
        popUpMsg("BAD SELECTION...Press OK")
      break
    endSwitch
  until (false or (LbBackup==true))
  // done
end

